# B&R Automation Studio project Teknologia25 (part 7)

### global.typ
```iecst
(*
Program: Robot

Description
(short summary)

*)
(*========== STATES ==========*)

TYPE
	RobotStateEnum :
		(
		ROBOT_INITIALIZE,
		ROBOT_IDLE,
		ROBOT_CMD_NORMAL,
		ROBOT_CMD_TARGET,
		ROBOT_COMMAND_DONE,
		ROBOT_COMMAND_ERROR,
		ROBOT_ERROR
		);
END_TYPE

(*========== INPUTS ==========*)

TYPE
	RobotInputCommandType : 	STRUCT
		Home : BOOL;
		PickUp : BOOL;
		GetCandy : BOOL;
		GiveCandy : BOOL;
		Dance : BOOL;
		HardReset : BOOL;
	END_STRUCT;
	RobotInputStatusType : 	STRUCT
		SetupComplete : BOOL;
	END_STRUCT;
	RobotInputType : 	STRUCT
		Force : BOOL;
		Command : RobotInputCommandType;
		Status : RobotInputStatusType;
		RobCommandNum : REAL;
		RobTargetX : REAL;
		RobTargetY : REAL;
	END_STRUCT;
END_TYPE

(*========== OUTPUTS ==========*)

TYPE
	RobotOutputCommandType : 	STRUCT
		NewCommand : BOOL;
	END_STRUCT;
	RobotOutputStatusType : 	STRUCT
		CommunicationOk : BOOL;
		CommandDone : BOOL;
		CommandError : BOOL;
		HardResetDone : BOOL;
		RobReady : BOOL;
		RobPhaseDone : BOOL;
		RobError : BOOL;
		RobPhaseNum : REAL;
		RobRapidState : BrAbbRwsStateRapidStateEnum;
		RobMotorState : BrAbbRwsStateMotorStateEnum;
		RobActiveMode : BrAbbRwsStateActiveModeEnum;
		ReadyForNextCommand : BOOL;
	END_STRUCT;
	RobotOutputType : 	STRUCT
		Command : RobotOutputCommandType;
		Status : RobotOutputStatusType;
	END_STRUCT;
END_TYPE

(*========== ERRORS ==========*)

TYPE
	RobotErrorType : 	STRUCT
		Active : BOOL;
		Acknowledge : BOOL;
		Code : DINT;
		Description : STRING[80];
	END_STRUCT;
END_TYPE

(*========== SETTINGS ==========*)

TYPE
	RobotSettingsType : 	STRUCT
		Enable : BOOL;
	END_STRUCT;
END_TYPE

(*========== INTERFACE ==========*)

TYPE
	RobotType : 	STRUCT
		Error : RobotErrorType;
		Input : RobotInputType;
		Output : RobotOutputType;
		Settings : RobotSettingsType;
		IsSimulated : BOOL;
		State : RobotStateEnum;
		SubState : DINT;
		StateInfo : STRING[255];
		OnStateEntry : BOOL; (*True for one cycle after state change*)
		robReadState : DINT;
	END_STRUCT;
END_TYPE
```

### Program Logical/Robot/Robot (IEC)

#### Robot.st
```iecst
PROGRAM _INIT

    // Access the task interface
	task ACCESS ADR(gRobot);

	// Check for simulator
	task.IsSimulated := DiagCpuIsSimulated();

	fb.BrAbbRwsCore_0.Parameters.UserName := 'Admin';
	fb.BrAbbRwsCore_0.Parameters.Password := 'robotics';
	fb.BrAbbRwsCore_0.Parameters.WebServerVersion := BR_ABB_RWS_VERSION_V2;
	fb.BrAbbRwsCore_0.Parameters.HostPort := 443;
	fb.BrAbbRwsCore_0.Parameters.Timeout := 0;
	fb.BrAbbRwsCore_0.Parameters.SecureConfigName := 'mySSLConfig';

	IF DiagCpuIsSimulated() THEN
		fb.BrAbbRwsCore_0.Parameters.ServerIP := '127.0.0.1';
	ELSE
		fb.BrAbbRwsCore_0.Parameters.ServerIP := '192.168.125.1';
	END_IF;

	fb.BrAbbRwsVariable_read.Parameters.Module := 'TeknologiaDemo25';
	fb.BrAbbRwsVariable_read.Parameters.Task := 'T_ROB1';
	fb.BrAbbRwsVariable_write.Parameters.Module := 'TeknologiaDemo25';
	fb.BrAbbRwsVariable_write.Parameters.Task := 'T_ROB1';

END_PROGRAM

PROGRAM _CYCLIC

    // Access task interface
    // =================================================================================================================
    task ACCESS ADR(gRobot);

    // Inputs
    // =================================================================================================================
    IF NOT task.Input.Force THEN
		task.Input.Command.Home := gMain.Output.Command.robHome;
		task.Input.Command.GetCandy := gMain.Output.Command.robGetPrize;
		task.Input.Command.Dance := gMain.Output.Command.robDance;
		task.Input.Command.GiveCandy := gMain.Output.Command.robGivePrize;
		task.Input.Command.PickUp := gMain.Output.Command.robPickup;
	END_IF

	task.Error.Active := fb.BrAbbRwsCore_0.Error OR fb.BrAbbRwsGetState_0.Error;

    // Task state machine
    // =================================================================================================================
    CASE task.State OF
        ROBOT_INITIALIZE:
			CASE task.SubState OF
				0:
					task.StateInfo := 'Initializing';
					// ---------------------------------------------------------------------------------
					fb.BrAbbRwsCore_0.Enable := FALSE;
					brsmemset(ADR(local), 0, SIZEOF(local));
					task.SubState := 10;
				10:
					task.StateInfo := 'Connecting to robot';
					// ---------------------------------------------------------------------------------
					fb.BrAbbRwsCore_0.Enable := TRUE;

					IF fb.BrAbbRwsCore_0.Active THEN
						task.State := ROBOT_IDLE;
						fb.BrAbbRwsGetState_0.Ident := fb.BrAbbRwsCore_0.Ident;
						fb.BrAbbRwsVariable_read.Ident := fb.BrAbbRwsCore_0.Ident;
						fb.BrAbbRwsVariable_write.Ident := fb.BrAbbRwsCore_0.Ident;
						local.readRobotValues := TRUE;
						fb.BrAbbRwsVariable_write.Enable := TRUE;
					ELSIF fb.BrAbbRwsCore_0.Error THEN
						task.Error.Code := fb.BrAbbRwsCore_0.StatusID;
						task.SubState := 30;
					END_IF;
			END_CASE;

		ROBOT_IDLE:
			task.StateInfo := 'Ready for commands';
			// ---------------------------------------------------------------------------------
			IF task.Input.Command.Home THEN
				task.Input.RobCommandNum := 1;
				task.State := ROBOT_CMD_NORMAL;

			ELSIF task.Input.Command.Dance THEN
				task.Input.RobCommandNum := 3;
				task.State := ROBOT_CMD_NORMAL;

			ELSIF task.Input.Command.GetCandy THEN
				task.Input.RobCommandNum := 4;
				task.State := ROBOT_CMD_NORMAL;

			ELSIF task.Input.Command.PickUp THEN
				task.Input.RobCommandNum := 2;
				task.State := ROBOT_CMD_TARGET;

			ELSIF task.Input.Command.GiveCandy THEN
				task.Input.RobCommandNum := 5;
				task.State := ROBOT_CMD_TARGET;
			END_IF;

		ROBOT_CMD_NORMAL:
			CASE task.SubState OF
				0:
					task.StateInfo := 'Execute command';
					// ---------------------------------------------------------------------------------
					fb.BrAbbRwsVariable_write.Parameters.Variable := 'nAcoposCmd';
					fb.BrAbbRwsVariable_write.Value.DataAdress := ADR(task.Input.RobCommandNum);
					fb.BrAbbRwsVariable_write.Value.DataType := BR_ABB_RWS_VAR_NUM;

					local.actions.substate.write := TRUE;

					IF fb.BrAbbRwsVariable_write.Done THEN
	  					task.SubState := 10;
					ELSIF fb.BrAbbRwsVariable_write.Error THEN
						task.State := ROBOT_COMMAND_ERROR;
					END_IF;

				10:
					task.StateInfo := 'Wait robot to complete';
					// ---------------------------------------------------------------------------------
					IF task.Output.Status.RobPhaseDone THEN
						task.SubState := 20;
					END_IF;

				20:
					task.StateInfo := 'Reset robot command';
					// ---------------------------------------------------------------------------------
					task.Input.RobCommandNum := 0;

					fb.BrAbbRwsVariable_write.Parameters.Variable := 'nAcoposCmd';
					fb.BrAbbRwsVariable_write.Value.DataAdress := ADR(task.Input.RobCommandNum);
					fb.BrAbbRwsVariable_write.Value.DataType := BR_ABB_RWS_VAR_NUM;

					local.actions.substate.write := TRUE;

					IF fb.BrAbbRwsVariable_write.Done THEN
						task.State := ROBOT_COMMAND_DONE;
					ELSIF fb.BrAbbRwsVariable_write.Error THEN
						task.State := ROBOT_COMMAND_ERROR;
					END_IF;
			END_CASE;

		ROBOT_CMD_TARGET:
			CASE task.SubState OF
				0:
					task.StateInfo := 'Write X';
					// ---------------------------------------------------------------------------------
					local.robTargetX_mm := 1000 * task.Input.RobTargetX;

					fb.BrAbbRwsVariable_write.Parameters.Variable := 'nPos_X';
					fb.BrAbbRwsVariable_write.Value.DataAdress := ADR(local.robTargetX_mm);
					fb.BrAbbRwsVariable_write.Value.DataType := BR_ABB_RWS_VAR_NUM;

					local.actions.substate.write := TRUE;

					IF fb.BrAbbRwsVariable_write.Done THEN
						task.SubState := 10;
					ELSIF fb.BrAbbRwsVariable_write.Error THEN
						task.State := ROBOT_COMMAND_ERROR;
					END_IF;

				10:
					task.StateInfo := 'Write Y';
					// ---------------------------------------------------------------------------------
					local.robTargetY_mm := 1000 * task.Input.RobTargetY;

					fb.BrAbbRwsVariable_write.Parameters.Variable := 'nPos_Y';
					fb.BrAbbRwsVariable_write.Value.DataAdress := ADR(local.robTargetY_mm);
					fb.BrAbbRwsVariable_write.Value.DataType := BR_ABB_RWS_VAR_NUM;

					local.actions.substate.write := TRUE;

					IF fb.BrAbbRwsVariable_write.Done THEN
						task.SubState := 20;
					ELSIF fb.BrAbbRwsVariable_write.Error THEN
						task.State := ROBOT_COMMAND_ERROR;
					END_IF;

				20:
					task.StateInfo := 'Write command num';
					// ---------------------------------------------------------------------------------
					fb.BrAbbRwsVariable_write.Parameters.Variable := 'nAcoposCmd';
					fb.BrAbbRwsVariable_write.Value.DataAdress := ADR(task.Input.RobCommandNum);
					fb.BrAbbRwsVariable_write.Value.DataType := BR_ABB_RWS_VAR_NUM;

					local.actions.substate.write := TRUE;

					IF fb.BrAbbRwsVariable_write.Done THEN
						task.SubState := 30;
					ELSIF fb.BrAbbRwsVariable_write.Error THEN
						task.State := ROBOT_COMMAND_ERROR;
					END_IF;

				30:
					task.StateInfo := 'Wait robot to complete';
					// ---------------------------------------------------------------------------------
					IF task.Output.Status.RobPhaseDone THEN
						task.SubState := 40;
					END_IF;

				40:
					task.StateInfo := 'Reset robot command';
					// ---------------------------------------------------------------------------------
					task.Input.RobCommandNum := 0;

					fb.BrAbbRwsVariable_write.Parameters.Variable := 'nAcoposCmd';
					fb.BrAbbRwsVariable_write.Value.DataAdress := ADR(task.Input.RobCommandNum);
					fb.BrAbbRwsVariable_write.Value.DataType := BR_ABB_RWS_VAR_NUM;

					local.actions.substate.write := TRUE;

					IF fb.BrAbbRwsVariable_write.Done THEN
						task.State := ROBOT_COMMAND_DONE;
					ELSIF fb.BrAbbRwsVariable_write.Error THEN
						task.State := ROBOT_COMMAND_ERROR;
					END_IF;
			END_CASE;

		ROBOT_COMMAND_DONE:
			task.StateInfo := 'Command done';
			// ---------------------------------------------------------------------------------
			local.actions.substate.command_done := TRUE;

			IF brsmemcmp(ADR(task.Input.Command), ADR(no_command), SIZEOF(no_command)) = 0 THEN
				task.State := ROBOT_IDLE;
			END_IF;

		ROBOT_COMMAND_ERROR:
			task.StateInfo := 'Command error';
			// ---------------------------------------------------------------------------------
			local.actions.substate.command_error := TRUE;
			local.actions.substate.write_reset := TRUE;

			IF brsmemcmp(ADR(task.Input.Command), ADR(no_command), SIZEOF(no_command)) = 0 THEN
				task.State := ROBOT_IDLE;
			END_IF;

		ROBOT_ERROR:
			// Error occured during execution
            // ---------------------------------------------------------------------------------
            IF task.Error.Acknowledge THEN
                brsmemset(ADR(task.Error), 0, SIZEOF(task.Error));
                task.State := ROBOT_INITIALIZE;
            END_IF;
    END_CASE // End of main task logic

    task.Error.Acknowledge := FALSE;

    // Detect state change events
    // =================================================================================================================
    task.OnStateEntry := (task.State <> local.lastState) OR (task.SubState <> local.lastSubState);

    IF task.State <> local.lastState THEN
        task.SubState := 0;
        local.lastState := task.State;
        brsmemset(ADR(local.actions.state), 0, SIZEOF(local.actions.state));
		brsmemset(ADR(local.actions.substate), 0, SIZEOF(local.actions.substate));
		task.StateInfo := '';
    END_IF

    // Reset current state actions also when substate changes
    IF task.SubState <> local.lastSubState THEN
        local.lastSubState := task.SubState;
		brsmemset(ADR(local.actions.substate), 0, SIZEOF(local.actions.substate));
		task.StateInfo := '';
    END_IF

	// Robot state poll
	// =================================================================================================================
	CASE task.robReadState OF
		0:
			// ---------------------------------------------------------------------------------
			IF local.readRobotValues THEN
				fb.BrAbbRwsGetState_0.Enable := TRUE;
				fb.BrAbbRwsVariable_read.Enable := TRUE;

				IF fb.BrAbbRwsGetState_0.Active AND fb.BrAbbRwsVariable_read.Active THEN

					task.robReadState := 10;
					local.robReadNum := 0;
				END_IF;
			END_IF;

		10:
			// ---------------------------------------------------------------------------------
			fb.TON_ReadDelay.IN := TRUE;
			fb.TON_ReadDelay.PT := T#20ms;

			IF local.readRobotValues = FALSE THEN
				task.robReadState := 0;
			ELSIF fb.TON_ReadDelay.Q THEN
				fb.TON_ReadDelay.IN := FALSE;
				task.robReadState := 100 + local.robReadNum;
				local.robReadNum := local.robReadNum + 1;
			END_IF;

		50:
			// ---------------------------------------------------------------------------------
			fb.TON_ReadDelay.IN := TRUE;
			fb.TON_ReadDelay.PT := T#2s;

			task.Output.Status.CommunicationOk := FALSE;

			fb.BrAbbRwsGetState_0.Enable := FALSE;
			fb.BrAbbRwsVariable_read.Enable := FALSE;

			IF fb.TON_ReadDelay.Q THEN
				fb.TON_ReadDelay.IN := FALSE;
				IF fb.BrAbbRwsCore_0.Error THEN
	  				task.robReadState := 60;
				ELSE
					task.robReadState := 0;
				END_IF;
			END_IF;

		60:
			// ---------------------------------------------------------------------------------
			fb.BrAbbRwsCore_0.ErrorReset := TRUE;

			IF NOT fb.BrAbbRwsCore_0.Error THEN
				fb.BrAbbRwsCore_0.ErrorReset := FALSE;
				task.robReadState := 0;
			END_IF;

		100:
			// ---------------------------------------------------------------------------------
			fb.BrAbbRwsGetState_0.Parameters.MechUnit := 'ROB1';
			fb.BrAbbRwsGetState_0.Parameters.Enable.ActPosCart := FALSE;
			fb.BrAbbRwsGetState_0.GetState := TRUE;

			IF fb.BrAbbRwsGetState_0.Done THEN
				task.Output.Status.CommunicationOk := TRUE;
				task.Output.Status.RobRapidState := fb.BrAbbRwsGetState_0.RapidState;
				task.Output.Status.RobMotorState := fb.BrAbbRwsGetState_0.MotorState;
				task.Output.Status.RobActiveMode := fb.BrAbbRwsGetState_0.ActiveMode;
				task.robReadState := 10;
			ELSIF fb.BrAbbRwsGetState_0.Error THEN
				task.Output.Status.RobRapidState := fb.BrAbbRwsGetState_0.RapidState;
				task.Output.Status.RobMotorState := fb.BrAbbRwsGetState_0.MotorState;
				task.Output.Status.RobActiveMode := fb.BrAbbRwsGetState_0.ActiveMode;
				task.robReadState := 50;
			END_IF;

		101:
			// ---------------------------------------------------------------------------------
			fb.BrAbbRwsVariable_read.Parameters.Variable := 'bRobotPhaseDone';
			fb.BrAbbRwsVariable_read.Value.DataAdress := ADR(gRobot.Output.Status.RobPhaseDone);
			fb.BrAbbRwsVariable_read.Value.DataType := BR_ABB_RWS_VAR_BOOL;
			fb.BrAbbRwsVariable_read.GetValue := TRUE;

			IF fb.BrAbbRwsVariable_read.Done THEN
				task.robReadState := 10;
			ELSIF fb.BrAbbRwsVariable_read.Error THEN
				task.robReadState := 50;
			END_IF;

		102:
			// ---------------------------------------------------------------------------------
			fb.BrAbbRwsVariable_read.Parameters.Variable := 'bRobotReady';
			fb.BrAbbRwsVariable_read.Value.DataAdress := ADR(gRobot.Output.Status.RobReady);
			fb.BrAbbRwsVariable_read.Value.DataType := BR_ABB_RWS_VAR_BOOL;
			fb.BrAbbRwsVariable_read.GetValue := TRUE;

			IF fb.BrAbbRwsVariable_read.Done THEN
				task.robReadState := 10;
			ELSIF fb.BrAbbRwsVariable_read.Error THEN
				task.robReadState := 50;
			END_IF;

		103:
			// ---------------------------------------------------------------------------------
			fb.BrAbbRwsVariable_read.Parameters.Variable := 'bRobotError';
			fb.BrAbbRwsVariable_read.Value.DataAdress := ADR(gRobot.Output.Status.RobError);
			fb.BrAbbRwsVariable_read.Value.DataType := BR_ABB_RWS_VAR_BOOL;
			fb.BrAbbRwsVariable_read.GetValue := TRUE;

			IF fb.BrAbbRwsVariable_read.Done THEN
				task.robReadState := 10;
			ELSIF fb.BrAbbRwsVariable_read.Error THEN
				task.robReadState := 50;
			END_IF;

		104:
			// ---------------------------------------------------------------------------------
			fb.BrAbbRwsVariable_read.Parameters.Variable := 'nRobotPhase';
			fb.BrAbbRwsVariable_read.Value.DataAdress := ADR(gRobot.Output.Status.RobPhaseNum);
			fb.BrAbbRwsVariable_read.Value.DataType := BR_ABB_RWS_VAR_NUM;
			fb.BrAbbRwsVariable_read.GetValue := TRUE;

			IF fb.BrAbbRwsVariable_read.Done THEN
				task.robReadState := 1000;
			ELSIF fb.BrAbbRwsVariable_read.Error THEN
				task.robReadState := 50;
			END_IF;

		1000:
			task.robReadState := 10;
			local.robReadNum := 0;
	END_CASE;

	IF task.robReadState <> local.robReadStateLast THEN
		local.robReadStateLast := task.robReadState;
		fb.BrAbbRwsGetState_0.GetState := FALSE;
		fb.BrAbbRwsVariable_read.GetValue := FALSE;
		fb.BrAbbRwsVariable_read.SetValue := FALSE;
		fb.BrAbbRwsVariable_read.SetValue := FALSE;
	END_IF;

    // Function calls
    // =================================================================================================================
    fb.BrAbbRwsCore_0();
	fb.TON_ReadDelay();
	fb.BrAbbRwsGetState_0();
	fb.BrAbbRwsVariable_read();

	fb.BrAbbRwsVariable_write.SetValue := local.actions.substate.write;
	fb.BrAbbRwsVariable_write.ErrorReset := local.actions.substate.write_reset;
	fb.BrAbbRwsVariable_write();

    // Task outputs
    // =================================================================================================================
	task.Output.Status.CommandDone := local.actions.substate.command_done;
	task.Output.Status.CommandError := local.actions.substate.command_error;

END_PROGRAM

PROGRAM _EXIT

//	WHILE fb.BrAbbRwsGetState_0.Active DO
//		fb.BrAbbRwsGetState_0(Enable := FALSE);
//	END_WHILE
//
//	WHILE fb.BrAbbRwsVariable_read.Active DO
//		fb.BrAbbRwsVariable_read(Enable := FALSE);
//	END_WHILE
//
//	task.robReadState := 100;
//	task.robReadState := 0;

END_PROGRAM
```

#### local.typ
```iecst
TYPE
	RobotFbType : 	STRUCT
		BrAbbRwsCore_0 : BrAbbRwsCore;
		BrAbbRwsVariable_read : BrAbbRwsVariable;
		BrAbbRwsVariable_write : BrAbbRwsVariable;
		BrAbbRwsGetState_0 : BrAbbRwsGetState;
		TON_RobState : TON;
		TON_ReadDelay : TON;
	END_STRUCT;
	RobotLocalType : 	STRUCT
		lastState : DINT;
		lastSubState : DINT;
		actions : RobotActionsType;
		readRobotValues : BOOL;
		robReadStateLast : DINT;
		robReadNum : DINT;
		robTargetX_mm : REAL;
		robTargetY_mm : REAL;
	END_STRUCT;
	RobotActionsType : 	STRUCT
		task : RobotTaskActionsType; (*Task actions are not automatically reset*)
		state : RobotStateActionsType; (*State actions are automatically reset whenever major task changes*)
		substate : RobotSubstateActionsType; (*Substate actions are automatically reset whenever major or substate changes*)
	END_STRUCT;
	RobotTaskActionsType : 	STRUCT
		task_action : BOOL;
	END_STRUCT;
	RobotStateActionsType : 	STRUCT
		state_action : BOOL;
	END_STRUCT;
	RobotSubstateActionsType : 	STRUCT
		command_done : BOOL;
		command_error : BOOL;
		write : BOOL;
		write_reset : BOOL;
	END_STRUCT;
	RobotHmiType : 	STRUCT
		isRunning : BOOL;
	END_STRUCT;
END_TYPE
```

#### local.var
```iecst
VAR
	task : REFERENCE TO RobotType;
	local : RobotLocalType;
	fb : RobotFbType;
	hmi : RobotHmiType;
	no_command : RobotInputCommandType;
END_VAR
```

- Visualisation Logical/mappView (not shown)

### Program Logical/Acp6D1 (IEC)

#### Acp6D.st
```iecst
PROGRAM _INIT

    // Access the task interface
	task ACCESS ADR(gAcp6D);

	// Check for simulator
	task.IsSimulated := DiagCpuIsSimulated();

	gCommInput;
	gCommOutput;
	gAssembly6D_1;

	// Fill in index of the shuttle element for easier access later on
	FOR i:=0 TO gMAX_INDEX_SHUTTLE DO
		local.shuttleOrder[i] := DINT_TO_UINT(i);
	END_FOR;

	acInitializePositions;

	moveQueueParamDefault.acceleration := 15.0;
	moveQueueParamDefault.acceleration_rotary := 0.1;
	moveQueueParamDefault.velocity_rotary := 0.1;
	moveQueueParamDefault.velocity_short := 0.1;
	moveQueueParamDefault.velocity_xy := 2.0;

	FOR i := 0 TO gMAX_INDEX_SHUTTLE DO
		fb.MoveQueue[i].Parameters := moveQueueParamDefault;
	END_FOR;

	// soundwave liikerata
	// Victory dance logiikka aalto z-aalto aalto -> vanhoihin asemmin -> keskellä spin ja z pomppuja -> kehällä arc movella kiertoradalle ja muutamak ierros ympäri -> paririviin keinahtelemaan ja kumartamaan pelaajalle
	// pelilogiikka mainiin
	// warm restartg mainiin
	// pelikäyttöliittymäsekvenssi
	// Circular shuffle loppuun -> group -> arc move -> sun planet -> asyncillä user selectiin
	// group fbt ja komennot
	// sun plenet tarkistus ja fb

END_PROGRAM

PROGRAM _CYCLIC
    // Access task interface
    // =================================================================================================================
	task ACCESS ADR(gAcp6D);

	test.SunShuttle := ADR(shuttles[4].Ref);
	test.PlanetShuttles[0] := shuttles[3].Ref;
	test();

	// Inputs
	// =================================================================================================================
	IF NOT task.Input.Force THEN
		task.Input.Command.MoveTo.Home := gMain.Output.Command.br6dHome;
		task.Input.Command.Shuffle.Circular := gMain.Output.Command.br6dcircularShuffle;
		task.Input.Command.FindPayload := gMain.Output.Command.br6dFindPayload;
		task.Input.Command.Victory := gMain.Output.Command.br6dLoseDance;
		task.Input.Command.ForceReset := gMain.Output.Command.br6dReset;
		task.Input.Command.SelectShuttle := gMain.Output.Command.br6dSelectShuttle;
		task.Input.Command.Shuffle.Simple := gMain.Output.Command.br6dSimpleShuffle;
		task.Input.Command.Victory := gMain.Output.Command.br6dWinDance;
	END_IF

	// Task state machine
	// =================================================================================================================
	CASE task.State OF
		ACP6D_INITIALIZE:
			CASE task.SubState OF
				0:
					task.StateInfo := 'Wait assembly to boot up';
					// ---------------------------------------------------------------------------------
					local.actions.state.cyclicModeRequest := a6dCYCLIC_DISABLED;

					fb.AssemblyReadInfo.Enable := TRUE;
					//Wait for the startup phase to be finished
					IF fb.AssemblyReadInfo.Valid THEN
						IF (fb.AssemblyReadInfo.AssemblyInfo.AssemblyState = mcACP6D_ERRORSTOP) THEN
							task.State := ACP6D_ERROR;
						ELSIF (fb.AssemblyReadInfo.AssemblyInfo.AssemblyState <> mcACP6D_STARTUP) THEN
							task.SubState := 10;
						END_IF
					END_IF

				10:
					task.StateInfo := 'Power off assembly';
					// ---------------------------------------------------------------------------------
					local.actions.substate.assemblyPowerOff := TRUE;

					IF fb.AssemblyPowerOff.Done THEN
						task.SubState := 20;
					ELSIF fb.AssemblyPowerOff.Error THEN
						task.Error.Code := fb.AssemblyPowerOff.ErrorID;
						task.State := ACP6D_ERROR;
					END_IF

				20:
					task.StateInfo := 'Power on assembly';
					// ---------------------------------------------------------------------------------
					IF task.OnStateEntry THEN
						brsmemset(ADR(shuttles), 0, SIZEOF(shuttles));
					END_IF;

					local.actions.substate.assemblyPowerOn := TRUE;

					IF fb.AssemblyPowerOn.Done THEN
						task.SubState := 100;
					ELSIF fb.AssemblyPowerOn.Error THEN
						task.Error.Code := fb.AssemblyPowerOn.ErrorID;
						task.State := ACP6D_ERROR;
					END_IF

				100:
					task.StateInfo := 'Read shuttle info - Read';
					// ---------------------------------------------------------------------------------
					local.actions.state.assemblyGetShuttles := TRUE;

					IF fb.AssemblyGetShuttle.Valid THEN
						task.Output.TotalShuttleCount := fb.AssemblyGetShuttle.TotalCount;
						local.actions.state.assemblyGetNextShuttle := FALSE;

						IF (fb.AssemblyGetShuttle.TotalCount = 0) THEN
							task.SubState := 1000;
							RETURN;
						END_IF;

						// Read shuttle information
						// Prevent access to wrong memory area
						i := LIMIT(0, UINT_TO_DINT(fb.AssemblyGetShuttle.TotalCount - fb.AssemblyGetShuttle.RemainingCount - 1), gMAX_INDEX_SHUTTLE);

						shuttles[i].ID := fb.AssemblyGetShuttle.AdditionalInfo.ShuttleID;
						shuttles[i].Ref := fb.AssemblyGetShuttle.Shuttle;
						shuttles[i].index := i;

						task.SubState := 110;
					END_IF

				110:
					task.StateInfo := 'Read shuttle info - Get next';
					// ---------------------------------------------------------------------------------
					IF (fb.AssemblyGetShuttle.RemainingCount > 0) THEN
						local.actions.state.assemblyGetNextShuttle := TRUE;
						task.SubState := 100;
					ELSE
						IF local.virtualShuttleCount >= MAX_NUM_SHUTTLE_VIRTUAL THEN
	  						task.State := ACP6D_COMMAND_DONE;
						ELSE
							task.SubState := 200;
						END_IF;
					END_IF

				200:
					task.StateInfo := 'Create virtual shuttle';
					// ---------------------------------------------------------------------------------
					local.actions.substate.createShuttleVirtual := TRUE;

					IF fb.virtualShCreate.Done THEN
						shuttlesVirtual[local.virtualShuttleCount] := fb.virtualShCreate.VirtualShuttle;
						local.virtualShuttleCount := local.virtualShuttleCount + 1;
						task.SubState := 210;
					ELSIF fb.virtualShCreate.Error THEN
						task.Error.Code := fb.virtualShCreate.ErrorID;
						task.State := ACP6D_ERROR;
					END_IF

				210:
					task.StateInfo := 'Check if enough virtual shuttles have been created';
					// ---------------------------------------------------------------------------------
					IF local.virtualShuttleCount >= MAX_NUM_SHUTTLE_VIRTUAL THEN
						task.State := ACP6D_COMMAND_DONE;
					ELSE
						task.SubState := 200;
					END_IF;

				1000:
					task.StateInfo := 'No shuttles';
				// ---------------------------------------------------------------------------------

			END_CASE;

		ACP6D_IDLE:
			task.StateInfo := 'Waiting for command';
			task.Output.Status.Initialized := TRUE;

			IF task.Input.Command.Reinitialize THEN
				task.State := ACP6D_INITIALIZE;

			ELSIF task.Input.Command.StartDemoMode THEN
				task.State := ACP6D_DEMO;

			ELSIF task.Input.Command.FindPayload THEN
				task.State := ACP6D_FIND_PAYLOAD;

			ELSIF task.Input.Command.SelectShuttle THEN
				task.State := ACP6D_SELECT_SHUTTLE;

			ELSIF task.Input.Command.StopAll THEN
				task.State := ACP6D_STOP_ALL;

			ELSIF task.Input.Command.ForceReset THEN
				task.State := ACP6D_FORCE_RESET;

			ELSIF task.Input.Command.Victory THEN
				task.State := ACP6D_VICTORY;

			ELSIF task.Input.Command.Animate THEN
				task.State := ACP6D_ANIMATE;

				// Move commands
			ELSIF task.Input.Command.MoveTo.Home THEN
				local.targetPos := positions.home;
				task.State := ACP6D_MOVE_TO;

			ELSIF task.Input.Command.MoveTo.User THEN
				local.targetPos := positions.user;
				task.State := ACP6D_MOVE_TO;

			ELSIF task.Input.Command.MoveTo.Dance THEN
				local.targetPos := positions.dance;
				task.State := ACP6D_MOVE_TO;

			ELSIF task.Input.Command.MoveTo.Clockface THEN
				local.targetPos := positions.clockface;
				task.State := ACP6D_MOVE_TO;

			ELSIF task.Input.Command.MoveTo.Pickup THEN
				local.targetPos := positions.pickup;
				task.State := ACP6D_MOVE_TO;

			ELSIF task.Input.Command.MoveTo.Shuffle THEN
				local.targetPos := positions.shuffle;
				task.State := ACP6D_MOVE_TO;

			ELSIF task.Input.Command.MoveTo.Side THEN
				local.targetPos := positions.side;
				task.State := ACP6D_MOVE_TO;

			// Shuffle commands
			ELSIF task.Input.Command.Shuffle.Simple THEN
				task.State := ACP6D_SHUFFLE_SIMPLE;

			ELSIF task.Input.Command.Shuffle.Circular THEN
				task.State := ACP6D_SHUFFLE_CIRCULAR;
			END_IF;

		ACP6D_DEMO:
			task.StateInfo := 'Running Acopos 6D feature demo';
			// ---------------------------------------------------------------------------------
			IF task.Input.Command.StopDemoMode THEN
				/// ..... Tähän kohtaan sit oma käsittely ja kun on demo taas inaktiviisiena niin hyppy COMMAND_DONE stateen
//				//IF FEATUREMODE INACTIEV THEN
//					task.State := ACP6D_COMMAND_DONE;
//				END_IF
			END_IF;

			//task.Output.Status.DemoModeActive := // MIKÄLIE LOGIIKKA ET MILLON ON PÄÄLLÄ!

		ACP6D_STOP_ALL:
			task.StateInfo := 'Stopping all shuttles';
			// ---------------------------------------------------------------------------------
			local.actions.substate.assemblyStop := TRUE;

			IF fb.assemblyStop.Done THEN
				task.State := ACP6D_COMMAND_DONE;
			ELSIF fb.assemblyStop.Done THEN
				task.Error.Code := fb.assemblyStop.ErrorID;
				task.State := ACP6D_COMMAND_ERROR;
			END_IF;

		ACP6D_FORCE_RESET:
			task.StateInfo := 'Stopping all shuttles';
			// ---------------------------------------------------------------------------------
			local.actions.substate.assemblyStop := TRUE;

			IF fb.assemblyStop.Done THEN
				task.State := ACP6D_INITIALIZE;
			ELSIF fb.assemblyStop.Done THEN
				task.Error.Code := fb.assemblyStop.ErrorID;
				task.State := ACP6D_COMMAND_ERROR;
			END_IF;

		ACP6D_MOVE_TO:
			CASE task.SubState OF
				0:
					task.StateInfo := 'Make sure assembly in correct state';
					// ---------------------------------------------------------------------------------
					task.SubState := 10;

				10:
					task.StateInfo := 'Move shuttles to target position';
					// ---------------------------------------------------------------------------------
					IF task.OnStateEntry THEN
						brfiShuffle(ADR(local.shuttleOrder));

						// Configure shuttle targets
						fb.MoveInPlaneAsync.Parameters.Velocity := 2;
						fb.MoveInPlaneAsync.Parameters.Acceleration := 15;

						fb.MoveInPlaneAsync.Parameters.Mode := mcACP6D_SHUTTLE_SORTED;

						FOR i := 0 TO gMAX_INDEX_SHUTTLE DO
							x := local.shuttleOrder[i];

							fb.MoveInPlaneAsync.Parameters.AsyncPar[i].Shuttle := ADR(shuttles[i].Ref);
							fb.MoveInPlaneAsync.Parameters.AsyncPar[x].X := local.targetPos[i].X;
							fb.MoveInPlaneAsync.Parameters.AsyncPar[x].Y := local.targetPos[i].Y;
						END_FOR;
					END_IF;

					local.actions.substate.moveInPlaneAsync := TRUE;

					IF fb.MoveInPlaneAsync.Done THEN
						task.State := ACP6D_COMMAND_DONE;
					ELSIF fb.MoveInPlaneAsync.Error THEN
						task.Error.Code := fb.MoveInPlaneAsync.ErrorID;
						task.State := ACP6D_COMMAND_ERROR;
					END_IF;
			END_CASE;

		ACP6D_FIND_PAYLOAD:
			CASE task.SubState OF
				0:
					task.StateInfo := 'Initialize';
					// ---------------------------------------------------------------------------------
					// Wait a moment before starting the force reading process so the movement has totally stopped
					local.actions.substate.delay := TRUE;
					fb.TON_delay.PT := T#1s;

					local.actions.state.cyclicModeRequest := a6dCYCLIC_READ_FORCE;

					// Also wait until all force readings are valid
					IF fb.TON_delay.Q AND cyclic.allForceValuesValid THEN
						task.SubState := 20;
					END_IF;

				20:
					task.StateInfo := 'Calculcate average Fz for shuttles';
					// ---------------------------------------------------------------------------------
					IF task.OnStateEntry THEN
						local.measurement_index := 0;
						FOR i := 0 TO gMAX_INDEX_SHUTTLE DO
							shuttle ACCESS ADR(shuttles[i]);
							brsmemset(ADR(shuttle.force.readings), 0, SIZEOF(shuttle.force.readings));
						END_FOR;
					END_IF;

					// Check if enough measurements have been recorder already
					IF local.measurement_index >= gMAX_INDEX_MEASUREMENT THEN
						FOR i := 0 TO gMAX_INDEX_SHUTTLE DO
							shuttle ACCESS ADR(shuttles[i]);

							shuttle.force.Z_avg := 0;

							FOR x := 0 TO gMAX_INDEX_MEASUREMENT DO
								shuttle.force.Z_avg := shuttle.force.Z_avg + shuttle.force.readings[x].Fz;
							END_FOR;

							shuttle.force.Z_avg := shuttle.force.Z_avg / MEASUREMENT_COUNT;
						END_FOR;
						task.SubState := 30;

					ELSIF shuttles[0].force.readings[local.measurement_index].Fz <> fb.ReadCyclicForce[0].CyclicForce.Fz THEN
						// Wait for next new value until measurement index is increased
						// Assume all channels received updates when first index of the cyclic force function block has new values
						FOR i := 0 TO gMAX_INDEX_SHUTTLE DO
							// Record received force values
							shuttle ACCESS ADR(shuttles[i]);
							shuttle.force.readings[local.measurement_index] := fb.ReadCyclicForce[shuttle.index].CyclicForce;
						END_FOR;

						local.measurement_index := local.measurement_index + 1;
					END_IF;

				30:
					task.StateInfo := 'Find which shuttle holds the payload';
					// ---------------------------------------------------------------------------------
					IF task.OnStateEntry THEN
						local.Fz_highest := 0;
					END_IF;

					FOR i := 0 TO gMAX_INDEX_SHUTTLE DO
						shuttle ACCESS ADR(shuttles[i]);

						IF shuttle.force.Z_avg > local.Fz_highest THEN
							local.Fz_highest := shuttle.force.Z_avg;
							task.Output.ShuttleWithPayload.index := i;
						END_IF;
					END_FOR;

					task.SubState := 40;

				40:
					task.StateInfo := 'Indicate which has payload';
					// ---------------------------------------------------------------------------------
					shuttle ACCESS ADR(shuttles[task.Output.ShuttleWithPayload.index]);
					refMoveQueue ACCESS ADR(fb.MoveQueue[shuttle.index]);

					IF task.OnStateEntry THEN
						refMoveQueue.Parameters.acceleration := 10;
						refMoveQueue.Parameters.velocity_short := 0.02;
						refMoveQueue.Parameters.velocity_xy := 1.0;

						AddCommand6D_xyz(ADR(commandQueue), sZ, 0, 0, 0.001, 0, 0, 0, mcACP6D_MOVE_ABSOLUTE);
						AddCommand6D_xyz(ADR(commandQueue), sZ, 0, 0, 0.004, 0, 0, 0, mcACP6D_MOVE_ABSOLUTE);
						AddCommand6D_xyz(ADR(commandQueue), sZ, 0, 0, 0.001, 0, 0, 0, mcACP6D_MOVE_ABSOLUTE);
						AddCommand6D_xyz(ADR(commandQueue), sZ, 0, 0, 0.004, 0, 0, 0, mcACP6D_MOVE_ABSOLUTE);
						AddCommand6D_xyz(ADR(commandQueue), sZ, 0, 0, 0.001, 0, 0, 0, mcACP6D_MOVE_ABSOLUTE);
						AddCommand6D_xyz(ADR(commandQueue), sZ, 0, 0, 0.004, 0, 0, 0, mcACP6D_MOVE_ABSOLUTE);
						AddCommand6D_xyz(ADR(commandQueue), sZ, 0, 0, 0.001, 0, 0, 0, mcACP6D_MOVE_ABSOLUTE);
						AddCommand6D_xyz(ADR(commandQueue), sZ, 0, 0, 0.004, 0, 0, 0, mcACP6D_MOVE_ABSOLUTE);
						AddCommand6D_xyz(ADR(commandQueue), sZ, 0, 0, 0.001, 0, 0, 0, mcACP6D_MOVE_ABSOLUTE);
						AddCommand6D_xyz(ADR(commandQueue), sZ, 0, 0, 0.004, 0, 0, 0, mcACP6D_MOVE_ABSOLUTE);
						AddCommand6D_xyz(ADR(commandQueue), sZ, 0, 0, 0.001, 0, 0, 0, mcACP6D_MOVE_ABSOLUTE);

						refMoveQueue.Commands := commandQueue;
					END_IF;

					shuttle.command.moveQueue := TRUE;

					IF refMoveQueue.Done THEN
						task.State := ACP6D_COMMAND_DONE;
					ELSIF refMoveQueue.Error THEN
						task.Error.Code := refMoveQueue.ErrorID;
						task.State := ACP6D_COMMAND_ERROR;
					END_IF;
			END_CASE

		ACP6D_SELECT_SHUTTLE:
			CASE task.SubState OF
				0:
					task.StateInfo := 'Move shuttles to the front of the table';
					// ---------------------------------------------------------------------------------
					IF task.OnStateEntry THEN
						local.selectedCount := brfiShuttleSelect(ADR(shuttles), ADR(selected1), 0, 0.24, 1, 1);

						FOR i := 0 TO gMAX_INDEX_SHUTTLE DO
							fb.MoveQueue[i].Parameters.velocity_short := 0.05;
						END_FOR;

						AddCommand6D_wait(ADR(commandQueue), 0);

						AddCommand6D_xyz(ADR(commandQueue), sZ, 0, 0, 0.001, 0, 0, 0, mcACP6D_MOVE_ABSOLUTE);
						AddCommand6D_xyz(ADR(commandQueue), sZ, 0, 0, 0.004, 0, 0, 0, mcACP6D_MOVE_ABSOLUTE);
						AddCommand6D_xyz(ADR(commandQueue), sZ, 0, 0, 0.001, 0, 0, 0, mcACP6D_MOVE_ABSOLUTE);
						AddCommand6D_xyz(ADR(commandQueue), sZ, 0, 0, 0.004, 0, 0, 0, mcACP6D_MOVE_ABSOLUTE);
						AddCommand6D_xyz(ADR(commandQueue), sZ, 0, 0, 0.001, 0, 0, 0, mcACP6D_MOVE_ABSOLUTE);
						AddCommand6D_xyz(ADR(commandQueue), sZ, 0, 0, 0.004, 0, 0, 0, mcACP6D_MOVE_ABSOLUTE);
						AddCommand6D_xyz(ADR(commandQueue), sZ, 0, 0, 0.001, 0, 0, 0, mcACP6D_MOVE_ABSOLUTE);

						AddCommand6D_xy(ADR(commandQueue), sY, 0, 0.900, 0, 0, 0, pathDIRECT, 0, mcACP6D_MOVE_ABSOLUTE);

						AddCommand6D_xyz(ADR(commandQueue), sZ, 0, 0, 0.003, 0, 0.1, 0, mcACP6D_MOVE_ABSOLUTE);
						AddCommand6D_Rxyz(ADR(commandQueue), sRx, -0.03, 0, 0, 0.3, mcACP6D_MOVE_ABSOLUTE);
						AddCommand6D_Rxyz(ADR(commandQueue), sRx, 0.00, 0, 0, 0.3, mcACP6D_MOVE_ABSOLUTE);

						AddCommand6D_xyz(ADR(commandQueue), sZ, 0, 0, 0.001, 0, 0, 0, mcACP6D_MOVE_ABSOLUTE);

						IF local.selectedCount > 0 THEN
							FOR i := 0 TO local.selectedCount - 1 DO
								fb.MoveQueue[selected1[i].index].Commands := commandQueue;
								fb.MoveQueue[selected1[i].index].Commands[0].waitTime := random.delays[i];
								shuttles[selected1[i].index].command.moveQueue := TRUE;
							END_FOR;
						END_IF;
					END_IF;

					IF queueStatus.allDone THEN
						task.SubState := 10;
					ELSIF queueStatus.error THEN
						task.Error.Code := queueStatus.errorID;
						task.State := ACP6D_COMMAND_ERROR;
					END_IF;

				10:
					task.StateInfo := 'Say hello to the player';
					// ---------------------------------------------------------------------------------
					IF task.OnStateEntry THEN
	  					local.selectedCount := brfiShuttleSelect(ADR(shuttles), ADR(selected1), 1, 1, 0, 0.240 * 3);

						AddCommand6D_wait(ADR(commandQueue), 0);
						AddCommand6D_xyz(ADR(commandQueue), sZ, 0, 0, 0.001, 0, 0, 0, mcACP6D_MOVE_ABSOLUTE);
						AddCommand6D_xyz(ADR(commandQueue), sZ, 0, 0, 0.004, 0, 0, 0, mcACP6D_MOVE_ABSOLUTE);
						AddCommand6D_wait(ADR(commandQueue), 0.1);
						AddCommand6D_xyz(ADR(commandQueue), sZ, 0, 0, 0.001, 0, 0, 0, mcACP6D_MOVE_ABSOLUTE);

						IF local.selectedCount > 0 THEN
							FOR i := 0 TO local.selectedCount - 1 DO
								fb.MoveQueue[selected1[i].index].Parameters.velocity_short := 0.03;

								fb.MoveQueue[selected1[i].index].Commands := commandQueue;
								fb.MoveQueue[selected1[i].index].Commands[0].waitTime := i * 0.1;
								shuttles[selected1[i].index].command.moveQueue := TRUE;
							END_FOR;
						END_IF;
					END_IF;

					IF queueStatus.allDone THEN
						task.SubState := 20;
					ELSIF queueStatus.error THEN
						task.Error.Code := queueStatus.errorID;
						task.State := ACP6D_COMMAND_ERROR;
					END_IF;

				20:
					task.StateInfo := 'Start force reading';
					// ---------------------------------------------------------------------------------
					local.actions.state.cyclicModeRequest := a6dCYCLIC_READ_FORCE;

					IF cyclic.allForceValuesValid THEN
						task.SubState := 30;
					END_IF;

				30:
					task.StateInfo := 'Wait user to select shuttle';
					// ---------------------------------------------------------------------------------
					IF task.OnStateEntry THEN
						FOR i := 0 TO gMAX_INDEX_SHUTTLE DO
							shuttle ACCESS ADR(shuttles[i]);
							shuttle.force.Fz_baseline := shuttle.force.value.Fz;
						END_FOR;
					END_IF

					FOR i := 0 TO gMAX_INDEX_SHUTTLE DO
						shuttle ACCESS ADR(shuttles[i]);
						// Detect shuttle press from force increase over treshold from baseline
						IF shuttle.force.value.Fz > (shuttle.force.Fz_baseline + 3.0) THEN
							task.SubState := 40;
							task.Output.ShuttleUserSelected.index := i;
						END_IF;
					END_FOR;

				40:
					task.StateInfo := 'Move selected shuttle';
					// ---------------------------------------------------------------------------------
					IF task.OnStateEntry THEN
						shuttle ACCESS ADR(shuttles[task.Output.ShuttleUserSelected.index]);
						refMoveQueue ACCESS ADR(fb.MoveQueue[shuttle.index]);

						refMoveQueue.Parameters.velocity_xy := 1.5;
						refMoveQueue.Parameters.acceleration := 5.0;

						AddCommand6D_xy(ADR(commandQueue), sX + sY, 0.0, -0.2, 0.5, 0.5, 0, pathDIRECT, 0, mcACP6D_MOVE_RELATIVE);
						AddCommand6D_xy(ADR(commandQueue), sX + sY, positions.pickup[0].X, positions.pickup[0].Y, 0, 15, 0, pathDIRECT, 0, mcACP6D_MOVE_ABSOLUTE);

						refMoveQueue.Commands := commandQueue;

						shuttle.command.moveQueue := TRUE;
					END_IF;

					IF refMoveQueue.Done THEN
						task.SubState := 50;
					ELSIF refMoveQueue.Error THEN
						task.Error.Code := refMoveQueue.ErrorID;
						task.SubState := ACP6D_COMMAND_ERROR;
					END_IF;

				50:
					task.StateInfo := 'Move all other shuttles to pickup';
					// ---------------------------------------------------------------------------------
					IF task.OnStateEntry THEN
						// Configure shuttle targets
						fb.MoveInPlaneAsync.Parameters.Velocity := 2;
						fb.MoveInPlaneAsync.Parameters.Acceleration := 15;

						fb.MoveInPlaneAsync.Parameters.Mode := mcACP6D_SHUTTLE_UNSORTED;

						x := 1;

						FOR i := 0 TO gMAX_INDEX_SHUTTLE DO
							IF i <> task.Output.ShuttleUserSelected.index THEN
								fb.MoveInPlaneAsync.Parameters.AsyncPar[i].Shuttle := ADR(shuttles[i].Ref);
								fb.MoveInPlaneAsync.Parameters.AsyncPar[i].X := positions.pickup[x].X;
								fb.MoveInPlaneAsync.Parameters.AsyncPar[i].Y := positions.pickup[x].Y;
								x := x + 1;
							END_IF;
						END_FOR;
					END_IF;

					local.actions.substate.moveInPlaneAsync := TRUE;

					IF fb.MoveInPlaneAsync.Done THEN
						task.SubState := 100;
					ELSIF fb.MoveInPlaneAsync.Error THEN
						task.Error.Code := fb.MoveInPlaneAsync.ErrorID;
						task.State := ACP6D_COMMAND_ERROR;
					END_IF;

				100:
					task.StateInfo := 'Transfer back to reading position values';
					// ---------------------------------------------------------------------------------
					local.actions.state.cyclicModeRequest := a6dCYCLIC_READ_POSITION;

					IF cyclic.allPositionsValid THEN
						task.State := ACP6D_COMMAND_DONE;
					END_IF;

			END_CASE;

		ACP6D_SHUFFLE_SIMPLE:
			CASE task.SubState OF
				0:
					task.StateInfo := 'Move shuttles to start position';
					// ---------------------------------------------------------------------------------
					IF task.OnStateEntry THEN
						brfiShuffle(ADR(local.shuttleOrder));

						brsmemset(ADR(shuffle), 0, SIZEOF(shuffle));

						// Configure shuttle targets
						fb.MoveInPlaneAsync.Parameters.Velocity := 2;
						fb.MoveInPlaneAsync.Parameters.Acceleration := 15;

						fb.MoveInPlaneAsync.Parameters.Mode := mcACP6D_SHUTTLE_SORTED;

						FOR i := 0 TO gMAX_INDEX_SHUTTLE DO
							x := local.shuttleOrder[i];
							IF x = shuttles[task.Output.ShuttleWithPayload.index].index THEN
	  							shuffle.payloadPos := i;
							END_IF;

							fb.MoveInPlaneAsync.Parameters.AsyncPar[i].Shuttle := ADR(shuttles[x].Ref);
							fb.MoveInPlaneAsync.Parameters.AsyncPar[i].X := positions.shuffle_simple[i].X;
							fb.MoveInPlaneAsync.Parameters.AsyncPar[i].Y := positions.shuffle_simple[i].Y;
						END_FOR;

						shuffle.randNum := RandValueDINT(0, 3);

						IF shuffle.payloadPos > 3 THEN
							fb.MoveInPlaneAsync.Parameters.AsyncPar[shuffle.payloadPos].Shuttle := fb.MoveInPlaneAsync.Parameters.AsyncPar[shuffle.randNum].Shuttle;
							fb.MoveInPlaneAsync.Parameters.AsyncPar[shuffle.randNum].Shuttle := ADR(shuttles[task.Output.ShuttleWithPayload.index].Ref);
						END_IF;

					END_IF;

					local.actions.substate.moveInPlaneAsync := TRUE;

					IF fb.MoveInPlaneAsync.Done THEN
						task.SubState := 10;
					ELSIF fb.MoveInPlaneAsync.Error THEN
						task.Error.Code := fb.MoveInPlaneAsync.ErrorID;
						task.State := ACP6D_COMMAND_ERROR;
					END_IF;

				10:
					task.StateInfo := 'Prepare for shuffle';
					// ---------------------------------------------------------------------------------
					brfiShuttleSelect(ADR(shuttles), ADR(selected1), 0, 0.480, 1, 1);
					fb.MoveQueue[selected1[0].index].Parameters := moveQueueParamDefault;
					fb.MoveQueue[selected1[1].index].Parameters := moveQueueParamDefault;
					fb.MoveQueue[selected1[2].index].Parameters := moveQueueParamDefault;
					fb.MoveQueue[selected1[3].index].Parameters := moveQueueParamDefault;
					shuffle.sequence := random.shuffleSequence;
					task.SubState := 20;

				20:
					task.StateInfo := 'Select next shuffle sequence';
					// ---------------------------------------------------------------------------------
					IF shuffle.step > gMAX_INDEX_SHUFFLE THEN
						task.SubState := 200;
					ELSE
						shuffle.invertedMove := shuffle.sequence[shuffle.step] < 0;
						shuffle.invertedDirection := SEL(shuffle.invertedMove, 1, -1);
						task.SubState := 100 + ABS(shuffle.sequence[shuffle.step]);
						shuffle.step := shuffle.step + 1;
					END_IF;

				100:
					task.StateInfo := 'Sides shift rotate';
					// ---------------------------------------------------------------------------------
					IF task.OnStateEntry THEN
						brfiShuttleSelect(ADR(shuttles), ADR(selected1), 0, 0.480, 1, 1);

						IF shuffle.invertedMove THEN
							AddCommand6D_arcAngularCW(ADR(fb.MoveQueue[selected1[0].index].Commands),  0.12, 0, brmPI, 0, 10, 0, mcACP6D_MOVE_RELATIVE);
							AddCommand6D_arcAngularCW(ADR(fb.MoveQueue[selected1[1].index].Commands), -0.12, 0, brmPI, 0, 10, 0, mcACP6D_MOVE_RELATIVE);

							AddCommand6D_arcAngularCW(ADR(fb.MoveQueue[selected1[2].index].Commands), 0.12, 0, brmPI, 0, 10, 0, mcACP6D_MOVE_RELATIVE);
							AddCommand6D_arcAngularCW(ADR(fb.MoveQueue[selected1[3].index].Commands), -0.12, 0, brmPI, 0, 10, 0, mcACP6D_MOVE_RELATIVE);
						ELSE
							AddCommand6D_arcAngularCCW(ADR(fb.MoveQueue[selected1[0].index].Commands),  0.12, 0, brmPI, 0, 10, 0, mcACP6D_MOVE_RELATIVE);
							AddCommand6D_arcAngularCCW(ADR(fb.MoveQueue[selected1[1].index].Commands), -0.12, 0, brmPI, 0, 10, 0, mcACP6D_MOVE_RELATIVE);

							AddCommand6D_arcAngularCCW(ADR(fb.MoveQueue[selected1[2].index].Commands), 0.12, 0, brmPI, 0, 10, 0, mcACP6D_MOVE_RELATIVE);
							AddCommand6D_arcAngularCCW(ADR(fb.MoveQueue[selected1[3].index].Commands), -0.12, 0, brmPI, 0, 10, 0, mcACP6D_MOVE_RELATIVE);
						END_IF;
					END_IF;

					shuttles[selected1[0].index].command.moveQueue := TRUE;
					shuttles[selected1[1].index].command.moveQueue := TRUE;
					shuttles[selected1[2].index].command.moveQueue := TRUE;
					shuttles[selected1[3].index].command.moveQueue := TRUE;

					IF queueStatus.allDone THEN
						task.SubState := 20;
					ELSIF queueStatus.error THEN
						task.Error.Code := queueStatus.errorID;
						task.State := ACP6D_COMMAND_ERROR;
					END_IF;

				101:
					task.StateInfo := 'Mid shift rotate';
					// ---------------------------------------------------------------------------------
					IF task.OnStateEntry THEN
						brfiShuttleSelect(ADR(shuttles), ADR(selected1), 0, 0.480, 1, 1);

						IF shuffle.invertedMove THEN
							AddCommand6D_arcAngularCW(ADR(commandQueue), 2 * 0.24, 3 * 0.24, brmPI, 0, 10, 0, mcACP6D_MOVE_ABSOLUTE);

							fb.MoveQueue[selected1[1].index].Commands := commandQueue;
							fb.MoveQueue[selected1[2].index].Commands := commandQueue;
						ELSE
							AddCommand6D_arcAngularCCW(ADR(commandQueue), 2 * 0.24, 3 * 0.24, brmPI, 0, 10, 0, mcACP6D_MOVE_ABSOLUTE);

							fb.MoveQueue[selected1[1].index].Commands := commandQueue;
							fb.MoveQueue[selected1[2].index].Commands := commandQueue;
						END_IF;
					END_IF;

					shuttles[selected1[1].index].command.moveQueue := TRUE;
					shuttles[selected1[2].index].command.moveQueue := TRUE;

					IF queueStatus.allDone THEN
						task.SubState := 20;
					ELSIF queueStatus.error THEN
						task.Error.Code := queueStatus.errorID;
						task.State := ACP6D_COMMAND_ERROR;
					END_IF;

				102:
					task.StateInfo := 'Sides shift';
					// ---------------------------------------------------------------------------------
					IF task.OnStateEntry THEN
						brfiShuttleSelect(ADR(shuttles), ADR(selected1), 0, 0.480, 1, 1);

						AddCommand6D_xy(ADR(fb.MoveQueue[selected1[0].index].Commands), sX + sY, 0, shuffle.invertedDirection  * -0.120, 0, 0, 0, pathY_X, 0, mcACP6D_MOVE_RELATIVE);
						AddCommand6D_xy(ADR(fb.MoveQueue[selected1[0].index].Commands), sX + sY, 3 * 0.240, 0, 0, 0, 0, pathY_X, 0, mcACP6D_MOVE_RELATIVE);
						AddCommand6D_xy(ADR(fb.MoveQueue[selected1[0].index].Commands), sX + sY, 0, shuffle.invertedDirection * 0.120, 0, 0, 0, pathY_X, 0, mcACP6D_MOVE_RELATIVE);

						AddCommand6D_xy(ADR(fb.MoveQueue[selected1[3].index].Commands), sX + sY, 0, shuffle.invertedDirection  * 0.120, 0, 0, 0, pathY_X, 0, mcACP6D_MOVE_RELATIVE);
						AddCommand6D_xy(ADR(fb.MoveQueue[selected1[3].index].Commands), sX + sY, -3 * 0.240, 0, 0, 0, 0, pathY_X, 0, mcACP6D_MOVE_RELATIVE);
						AddCommand6D_xy(ADR(fb.MoveQueue[selected1[3].index].Commands), sX + sY, 0, shuffle.invertedDirection  * -0.120, 0, 0, 0, pathY_X, 0, mcACP6D_MOVE_RELATIVE);
					END_IF;

					shuttles[selected1[0].index].command.moveQueue := TRUE;
					shuttles[selected1[3].index].command.moveQueue := TRUE;

					IF queueStatus.allDone THEN
						task.SubState := 20;
					ELSIF queueStatus.error THEN
						task.Error.Code := queueStatus.errorID;
						task.State := ACP6D_COMMAND_ERROR;
					END_IF;

				103:
					task.StateInfo := 'Middle to outside shift';
					// ---------------------------------------------------------------------------------
					IF task.OnStateEntry THEN
						brfiShuttleSelect(ADR(shuttles), ADR(selected1), 0, 0.480, 1, 1);

						AddCommand6D_xy(ADR(fb.MoveQueue[selected1[0].index].Commands), sX + sY, 0.240, 0, 0, 0, 0, pathY_X, 0.00, mcACP6D_MOVE_RELATIVE);
						AddCommand6D_xy(ADR(fb.MoveQueue[selected1[3].index].Commands), sX + sY, -0.240, 0, 0, 0, 0, pathY_X, 0.00, mcACP6D_MOVE_RELATIVE);

						AddCommand6D_xy(ADR(fb.MoveQueue[selected1[1].index].Commands), sX + sY, 0, shuffle.invertedDirection * 0.120, 0, 0, 0, pathY_X, 0.00, mcACP6D_MOVE_RELATIVE);
						AddCommand6D_xy(ADR(fb.MoveQueue[selected1[1].index].Commands), sX + sY, -0.240, 0, 0, 0, 0, pathY_X, 0.00, mcACP6D_MOVE_RELATIVE);
						AddCommand6D_xy(ADR(fb.MoveQueue[selected1[1].index].Commands), sX + sY, 0, shuffle.invertedDirection * -0.120, 0, 0, 0, pathY_X, 0.00, mcACP6D_MOVE_RELATIVE);

						AddCommand6D_xy(ADR(fb.MoveQueue[selected1[2].index].Commands), sX + sY, 0, shuffle.invertedDirection * 0.120, 0, 0, 0, pathY_X, 0.00, mcACP6D_MOVE_RELATIVE);
						AddCommand6D_xy(ADR(fb.MoveQueue[selected1[2].index].Commands), sX + sY, 0.240, 0, 0, 0, 0, pathY_X, 0.00, mcACP6D_MOVE_RELATIVE);
						AddCommand6D_xy(ADR(fb.MoveQueue[selected1[2].index].Commands), sX + sY, 0, shuffle.invertedDirection * -0.120, 0, 0, 0, pathY_X, 0.00, mcACP6D_MOVE_RELATIVE);
					END_IF;

					shuttles[selected1[0].index].command.moveQueue := TRUE;
					shuttles[selected1[1].index].command.moveQueue := TRUE;
					shuttles[selected1[2].index].command.moveQueue := TRUE;
					shuttles[selected1[3].index].command.moveQueue := TRUE;

					IF queueStatus.allDone THEN
						task.SubState := 20;
					ELSIF queueStatus.error THEN
						task.Error.Code := queueStatus.errorID;
						task.State := ACP6D_COMMAND_ERROR;
					END_IF;

				104:
					task.StateInfo := 'Twin shift';
					// ---------------------------------------------------------------------------------
					IF task.OnStateEntry THEN
						brfiShuttleSelect(ADR(shuttles), ADR(selected1), 0, 0.480, 1, 1);

						AddCommand6D_xy(ADR(fb.MoveQueue[selected1[0].index].Commands), sX + sY, 0, shuffle.invertedDirection * 0.120, 0, 0, 0, pathY_X, 0.00, mcACP6D_MOVE_RELATIVE);
						AddCommand6D_xy(ADR(fb.MoveQueue[selected1[2].index].Commands), sX + sY, 0, shuffle.invertedDirection * 0.120, 0, 0, 0, pathY_X, 0.00, mcACP6D_MOVE_RELATIVE);
						AddCommand6D_xy(ADR(fb.MoveQueue[selected1[0].index].Commands), sX + sY, 0.240, 0, 0, 0, 0, pathY_X, 0.00, mcACP6D_MOVE_RELATIVE);
						AddCommand6D_xy(ADR(fb.MoveQueue[selected1[2].index].Commands), sX + sY, 0.240, 0, 0, 0, 0, pathY_X, 0.00, mcACP6D_MOVE_RELATIVE);
						AddCommand6D_xy(ADR(fb.MoveQueue[selected1[0].index].Commands), sX + sY, 0, shuffle.invertedDirection * -0.120, 0, 0, 0, pathY_X, 0.00, mcACP6D_MOVE_RELATIVE);
						AddCommand6D_xy(ADR(fb.MoveQueue[selected1[2].index].Commands), sX + sY, 0, shuffle.invertedDirection * -0.120, 0, 0, 0, pathY_X, 0.00, mcACP6D_MOVE_RELATIVE);

						AddCommand6D_xy(ADR(fb.MoveQueue[selected1[1].index].Commands), sX + sY, 0, shuffle.invertedDirection * -0.120, 0, 0, 0, pathY_X, 0.00, mcACP6D_MOVE_RELATIVE);
						AddCommand6D_xy(ADR(fb.MoveQueue[selected1[3].index].Commands), sX + sY, 0, shuffle.invertedDirection * -0.120, 0, 0, 0, pathY_X, 0.00, mcACP6D_MOVE_RELATIVE);
						AddCommand6D_xy(ADR(fb.MoveQueue[selected1[1].index].Commands), sX + sY, -0.240, 0, 0, 0, 0, pathY_X, 0.00, mcACP6D_MOVE_RELATIVE);
						AddCommand6D_xy(ADR(fb.MoveQueue[selected1[3].index].Commands), sX + sY, -0.240, 0, 0, 0, 0, pathY_X, 0.00, mcACP6D_MOVE_RELATIVE);
						AddCommand6D_xy(ADR(fb.MoveQueue[selected1[1].index].Commands), sX + sY, 0, shuffle.invertedDirection * 0.120, 0, 0, 0, pathY_X, 0.00, mcACP6D_MOVE_RELATIVE);
						AddCommand6D_xy(ADR(fb.MoveQueue[selected1[3].index].Commands), sX + sY, 0, shuffle.invertedDirection * 0.120, 0, 0, 0, pathY_X, 0.00, mcACP6D_MOVE_RELATIVE);
					END_IF;

					shuttles[selected1[0].index].command.moveQueue := TRUE;
					shuttles[selected1[1].index].command.moveQueue := TRUE;
					shuttles[selected1[2].index].command.moveQueue := TRUE;
					shuttles[selected1[3].index].command.moveQueue := TRUE;

					IF queueStatus.allDone THEN
						task.SubState := 20;
					ELSIF queueStatus.error THEN
						task.Error.Code := queueStatus.errorID;
						task.State := ACP6D_COMMAND_ERROR;
					END_IF;

				200:
					task.StateInfo := 'Star shift 1';
					// ---------------------------------------------------------------------------------
					IF task.OnStateEntry THEN
						brfiShuttleSelect(ADR(shuttles), ADR(selected1), 0, 0.480, 1, 1);

						AddCommand6D_xy(ADR(fb.MoveQueue[selected1[0].index].Commands), sX + sY,  0.360, 0.140, 0, 0, 0, pathY_X, 0.00, mcACP6D_MOVE_RELATIVE);
						AddCommand6D_xy(ADR(fb.MoveQueue[selected1[3].index].Commands), sX + sY,  -0.360, -0.140, 0, 0, 0, pathY_X, 0.00, mcACP6D_MOVE_RELATIVE);

						AddCommand6D_xy(ADR(fb.MoveQueue[selected1[1].index].Commands), sX + sY,  -0.020, 0, 0, 0, 0, pathY_X, 0.00, mcACP6D_MOVE_RELATIVE);
						AddCommand6D_xy(ADR(fb.MoveQueue[selected1[2].index].Commands), sX + sY,  0.020, 0, 0, 0, 0, pathY_X, 0.00, mcACP6D_MOVE_RELATIVE);
					END_IF;

					shuttles[selected1[0].index].command.moveQueue := TRUE;
					shuttles[selected1[1].index].command.moveQueue := TRUE;
					shuttles[selected1[2].index].command.moveQueue := TRUE;
					shuttles[selected1[3].index].command.moveQueue := TRUE;

					IF queueStatus.allDone THEN
						task.SubState := 201;
					ELSIF queueStatus.error THEN
						task.Error.Code := queueStatus.errorID;
						task.State := ACP6D_COMMAND_ERROR;
					END_IF;

				201:
					task.StateInfo := 'Star shift 2';
					// ---------------------------------------------------------------------------------
					IF task.OnStateEntry THEN
						shuttle ACCESS ADR(shuttles[selected1[0].index]);

						shuffle.angle := brmPI_2 * RandValueDINT(3 * 4, 5 * 4);

						brsmemset(ADR(commandQueue), 0, SIZEOF(commandQueue));

						AddCommand6D_waitCmdLb(ADR(commandQueue), shuttle.ID, mcACP6D_SH_WAIT_CMDLB_START, 0, mcACP6D_SH_WAIT_CMDLB_REGULAR);
						AddCommand6D_arcAngularCW(ADR(commandQueue), 2 * 0.24, 3 * 0.24, shuffle.angle, 1.0, 15.0, 0, mcACP6D_MOVE_ABSOLUTE);

						fb.MoveQueue[selected1[1].index].Commands := commandQueue;
						fb.MoveQueue[selected1[2].index].Commands := commandQueue;
						fb.MoveQueue[selected1[3].index].Commands := commandQueue;
					END_IF;

					shuttles[selected1[1].index].command.moveQueue := TRUE;
					shuttles[selected1[2].index].command.moveQueue := TRUE;
					shuttles[selected1[3].index].command.moveQueue := TRUE;

					IF fb.MoveQueue[selected1[1].index].Acknowledge AND fb.MoveQueue[selected1[2].index].Acknowledge AND fb.MoveQueue[selected1[3].index].Acknowledge THEN
						task.SubState := 202;
					ELSIF queueStatus.error THEN
						task.Error.Code := queueStatus.errorID;
						task.State := ACP6D_COMMAND_ERROR;
					END_IF;

				202:
					task.StateInfo := 'Star shift 3';
					// ---------------------------------------------------------------------------------
					IF task.OnStateEntry THEN
						shuttle ACCESS ADR(shuttles[selected1[0].index]);

						AddCommand6D_arcAngularCW(ADR(commandQueue), 2 * 0.24, 3 * 0.24, shuffle.angle, 1.0, 15.0, 0, mcACP6D_MOVE_ABSOLUTE);

						fb.MoveQueue[selected1[0].index].Commands := commandQueue;
					END_IF;

					shuttles[selected1[0].index].command.moveQueue := TRUE;

					IF queueStatus.allDone THEN
						task.SubState := 203;
					ELSIF queueStatus.error THEN
						task.Error.Code := queueStatus.errorID;
						task.State := ACP6D_COMMAND_ERROR;
					END_IF;

				203:
					task.StateInfo := 'Star shift end';
					// ---------------------------------------------------------------------------------
					IF task.OnStateEntry THEN
						brfiShuttleSelect(ADR(shuttles), ADR(selected1), 0, 0.480, 1, 1);

						AddCommand6D_xy(ADR(fb.MoveQueue[selected1[0].index].Commands), sX + sY, positions.shuffle_simple[0].X, positions.shuffle_simple[0].Y, 0, 0, 0, pathDIRECT, 0.00, mcACP6D_MOVE_ABSOLUTE);
						AddCommand6D_xy(ADR(fb.MoveQueue[selected1[1].index].Commands), sX + sY, positions.shuffle_simple[1].X, positions.shuffle_simple[1].Y, 0, 0, 0, pathDIRECT, 0.00, mcACP6D_MOVE_ABSOLUTE);
						AddCommand6D_xy(ADR(fb.MoveQueue[selected1[2].index].Commands), sX + sY, positions.shuffle_simple[2].X, positions.shuffle_simple[2].Y, 0, 0, 0, pathDIRECT, 0.00, mcACP6D_MOVE_ABSOLUTE);
						AddCommand6D_xy(ADR(fb.MoveQueue[selected1[3].index].Commands), sX + sY, positions.shuffle_simple[3].X, positions.shuffle_simple[3].Y, 0, 0, 0, pathDIRECT, 0.00, mcACP6D_MOVE_ABSOLUTE);
					END_IF;

					shuttles[selected1[0].index].command.moveQueue := TRUE;
					shuttles[selected1[1].index].command.moveQueue := TRUE;
					shuttles[selected1[2].index].command.moveQueue := TRUE;
					shuttles[selected1[3].index].command.moveQueue := TRUE;

					IF queueStatus.allDone THEN
						task.SubState := 204;
					ELSIF queueStatus.error THEN
						task.Error.Code := queueStatus.errorID;
						task.State := ACP6D_COMMAND_ERROR;
					END_IF;

				204:
					task.StateInfo := 'End of simple shuffle - move to select';
					// ---------------------------------------------------------------------------------
					IF task.OnStateEntry THEN
						brfiShuttleSelect(ADR(shuttles), ADR(selected1), 0, 0.480, 1, 1);

						AddCommand6D_xy(ADR(fb.MoveQueue[selected1[0].index].Commands), sX + sY, positions.user[2].X, positions.user[2].Y, 1.5, 0, 0, pathDIRECT, 0.00, mcACP6D_MOVE_ABSOLUTE);
						AddCommand6D_xy(ADR(fb.MoveQueue[selected1[1].index].Commands), sX + sY, positions.user[3].X, positions.user[3].Y, 1.5, 0, 0, pathDIRECT, 0.00, mcACP6D_MOVE_ABSOLUTE);
						AddCommand6D_xy(ADR(fb.MoveQueue[selected1[2].index].Commands), sX + sY, positions.user[4].X, positions.user[4].Y, 1.5, 0, 0, pathDIRECT, 0.00, mcACP6D_MOVE_ABSOLUTE);
						AddCommand6D_xy(ADR(fb.MoveQueue[selected1[3].index].Commands), sX + sY, positions.user[5].X, positions.user[5].Y, 1.5, 0, 0, pathDIRECT, 0.00, mcACP6D_MOVE_ABSOLUTE);
					END_IF;

					shuttles[selected1[0].index].command.moveQueue := TRUE;
					shuttles[selected1[1].index].command.moveQueue := TRUE;
					shuttles[selected1[2].index].command.moveQueue := TRUE;
					shuttles[selected1[3].index].command.moveQueue := TRUE;

					IF queueStatus.allDone THEN
						task.State := ACP6D_COMMAND_DONE;
					ELSIF queueStatus.error THEN
						task.Error.Code := queueStatus.errorID;
						task.State := ACP6D_COMMAND_ERROR;
					END_IF;

			END_CASE;

		ACP6D_SHUFFLE_CIRCULAR:
			CASE task.SubState OF
				0:
					task.StateInfo := 'Move shuttles to start position';
					// ---------------------------------------------------------------------------------
					IF task.OnStateEntry THEN
						brfiShuffle(ADR(local.shuttleOrder));

						// Configure shuttle targets
						fb.MoveInPlaneAsync.Parameters.Velocity := 2;
						fb.MoveInPlaneAsync.Parameters.Acceleration := 15;

						fb.MoveInPlaneAsync.Parameters.Mode := mcACP6D_SHUTTLE_SORTED;

						FOR i := 0 TO gMAX_INDEX_SHUTTLE DO
							x := local.shuttleOrder[i];
							fb.MoveInPlaneAsync.Parameters.AsyncPar[i].Shuttle := ADR(shuttles[x].Ref);
							fb.MoveInPlaneAsync.Parameters.AsyncPar[i].X := positions.clockface[i].X;
							fb.MoveInPlaneAsync.Parameters.AsyncPar[i].Y := positions.clockface[i].Y;
						END_FOR;
					END_IF;

					local.actions.substate.moveInPlaneAsync := TRUE;

					IF fb.MoveInPlaneAsync.Done THEN
						task.SubState := 100;
					ELSIF fb.MoveInPlaneAsync.Error THEN
						task.Error.Code := fb.MoveInPlaneAsync.ErrorID;
						task.State := ACP6D_COMMAND_ERROR;
					END_IF;

				100:
					task.StateInfo := 'Add commands to queue';
					// ---------------------------------------------------------------------------------
					IF task.OnStateEntry THEN
						shuttle ACCESS ADR(shuttles[0]);

						shuffle.angle := (brmPI/8) * RandValueDINT(6 * 8, 9 * 8);

						brsmemset(ADR(commandQueue), 0, SIZEOF(commandQueue));

						AddCommand6D_waitCmdLb(ADR(commandQueue), shuttle.ID, mcACP6D_SH_WAIT_CMDLB_START, 0, mcACP6D_SH_WAIT_CMDLB_REGULAR);
						AddCommand6D_arcAngularCW(ADR(commandQueue), 0.48, 0.48, shuffle.angle, 0, 0, 0, mcACP6D_MOVE_ABSOLUTE);

						FOR i := 0 TO gMAX_INDEX_SHUTTLE DO
							fb.MoveQueue[i].Parameters := moveQueueParamDefault;
							fb.MoveQueue[i].Parameters.acceleration := 14.0;
						END_FOR;

						FOR i := 1 TO gMAX_INDEX_SHUTTLE DO
							fb.MoveQueue[i].Commands := commandQueue;
							shuttles[i].command.moveQueue := TRUE;
						END_FOR;
					END_IF

					IF queueStatus.allAcknowledge THEN
						task.SubState := 110;
					ELSIF queueStatus.error THEN
						task.Error.Code := queueStatus.errorID;
						task.State := ACP6D_COMMAND_ERROR;
					END_IF;

				110:
					task.StateInfo := 'Wait to finish circular CW';
					// ---------------------------------------------------------------------------------
					IF task.OnStateEntry THEN
						brsmemset(ADR(commandQueue), 0, SIZEOF(commandQueue));

						AddCommand6D_arcAngularCW(ADR(commandQueue), 0.48, 0.48, shuffle.angle, 0, 0, 0, mcACP6D_MOVE_ABSOLUTE);

						fb.MoveQueue[0].Commands := commandQueue;
						shuttles[0].command.moveQueue := TRUE;
					END_IF

					IF queueStatus.allDone THEN
						task.SubState := 120;
					ELSIF queueStatus.error THEN
						task.Error.Code := queueStatus.errorID;
						task.State := ACP6D_COMMAND_ERROR;
					END_IF;

				120:
					task.StateInfo := 'Add commands to queue';
					// ---------------------------------------------------------------------------------
					IF task.OnStateEntry THEN
						shuttle ACCESS ADR(shuttles[0]);

						shuffle.angle := (brmPI/8) * RandValueDINT(6 * 8, 9 * 8);

						brsmemset(ADR(commandQueue), 0, SIZEOF(commandQueue));

						AddCommand6D_waitCmdLb(ADR(commandQueue), shuttle.ID, mcACP6D_SH_WAIT_CMDLB_START, 0, mcACP6D_SH_WAIT_CMDLB_REGULAR);
						AddCommand6D_arcAngularCCW(ADR(commandQueue), 0.48, 0.48, shuffle.angle, 0, 0, 0, mcACP6D_MOVE_ABSOLUTE);

						FOR i := 1 TO gMAX_INDEX_SHUTTLE DO
							fb.MoveQueue[i].Commands := commandQueue;
							shuttles[i].command.moveQueue := TRUE;
						END_FOR;
					END_IF

					IF queueStatus.allAcknowledge THEN
						task.SubState := 130;
					ELSIF queueStatus.error THEN
						task.Error.Code := queueStatus.errorID;
						task.State := ACP6D_COMMAND_ERROR;
					END_IF;

				130:
					task.StateInfo := 'wait to finish circular CCW';
					// ---------------------------------------------------------------------------------
					IF task.OnStateEntry THEN
						brsmemset(ADR(commandQueue), 0, SIZEOF(commandQueue));

						AddCommand6D_arcAngularCCW(ADR(commandQueue), 0.48, 0.48, shuffle.angle, 0, 0, 0, mcACP6D_MOVE_ABSOLUTE);

						fb.MoveQueue[0].Commands := commandQueue;
						shuttles[0].command.moveQueue := TRUE;
					END_IF

					IF queueStatus.allDone THEN
						task.SubState := 200;
					ELSIF queueStatus.error THEN
						task.Error.Code := queueStatus.errorID;
						task.State := ACP6D_COMMAND_ERROR;
					END_IF;

				200:
					task.StateInfo := 'Move shuttles to kongo line';
					// ---------------------------------------------------------------------------------
					IF task.OnStateEntry THEN
						brfiShuffle(ADR(local.shuttleOrder));

						// Configure shuttle targets
						fb.MoveInPlaneAsync.Parameters.Velocity := 2;
						fb.MoveInPlaneAsync.Parameters.Acceleration := 15;

						fb.MoveInPlaneAsync.Parameters.Mode := mcACP6D_SHUTTLE_SORTED;

						FOR i := 0 TO gMAX_INDEX_SHUTTLE DO
							x := local.shuttleOrder[i];
							fb.MoveInPlaneAsync.Parameters.AsyncPar[i].Shuttle := ADR(shuttles[x].Ref);
							fb.MoveInPlaneAsync.Parameters.AsyncPar[i].X := positions.kongo_lines[i].X;
							fb.MoveInPlaneAsync.Parameters.AsyncPar[i].Y := positions.kongo_lines[i].Y;
						END_FOR;
					END_IF;

					local.actions.substate.moveInPlaneAsync := TRUE;

					IF fb.MoveInPlaneAsync.Done THEN
						task.SubState := 210;
					ELSIF fb.MoveInPlaneAsync.Error THEN
						task.Error.Code := fb.MoveInPlaneAsync.ErrorID;
						task.State := ACP6D_COMMAND_ERROR;
					END_IF;

				210:
					task.StateInfo := 'Move shuttles to start position';
					// ---------------------------------------------------------------------------------
					IF task.OnStateEntry THEN
						brfiShuttleSelect(ADR(shuttles), ADR(selected1), 0, 0, 2 * 0.240, 1);
						brfiShuttleSelect(ADR(shuttles), ADR(selected2), 2 * 0.240, 0, 1, 1);

						AddCommand6D_xy(ADR(commandQueue), sX, 0.240 + 0.120, 0, 0, 0, 1, pathDIRECT, 0, mcACP6D_MOVE_RELATIVE);
						AddCommand6D_arcAngularCCW(ADR(commandQueue), 0, 0.060, brmPI, 0, 0, 1, mcACP6D_MOVE_RELATIVE);
						AddCommand6D_xy(ADR(commandQueue), sX, -0.480, 0, 0, 0, 1, pathDIRECT, 0, mcACP6D_MOVE_RELATIVE);

						AddCommand6D_arcAngularCCW(ADR(commandQueue), 0, -0.060, brmPI, 0, 0, 1, mcACP6D_MOVE_RELATIVE);
						AddCommand6D_xy(ADR(commandQueue), sX, 0.120, 0, 0, 0, 1, pathDIRECT, 0, mcACP6D_MOVE_RELATIVE);
						AddCommand6D_xy(ADR(commandQueue), sX, 0.240 + 0.120, 0, 0, 0, 1, pathDIRECT, 0, mcACP6D_MOVE_RELATIVE);
						AddCommand6D_arcAngularCCW(ADR(commandQueue), 0, 0.060, brmPI, 0, 0, 1, mcACP6D_MOVE_RELATIVE);

						AddCommand6D_xy(ADR(commandQueue), sX, -0.480, 0, 0, 0, 1, pathDIRECT, 0, mcACP6D_MOVE_RELATIVE);
						AddCommand6D_arcAngularCCW(ADR(commandQueue), 0, -0.060, brmPI, 0, 0, 1, mcACP6D_MOVE_RELATIVE);
						AddCommand6D_xy(ADR(commandQueue), sX, 0.240 + 0.120, 0, 0, 0, 1, pathDIRECT, 0, mcACP6D_MOVE_RELATIVE);
						AddCommand6D_arcAngularCCW(ADR(commandQueue), 0, 0.060, brmPI, 0, 0, 1, mcACP6D_MOVE_RELATIVE);

						AddCommand6D_xy(ADR(commandQueue), sX, 2 * 0.240, 0, 0, 0, 0, pathDIRECT, 0, mcACP6D_MOVE_ABSOLUTE);

						FOR i := 0 TO 3 DO
							fb.MoveQueue[selected1[i].index].Commands := commandQueue;
							shuttles[selected1[i].index].command.moveQueue := TRUE;;
						END_FOR;

						brsmemset(ADR(commandQueue), 0, SIZEOF(commandQueue));
						AddCommand6D_xy(ADR(commandQueue), sX, -(0.240 + 0.120), 0, 0, 0, 1, pathDIRECT, 0, mcACP6D_MOVE_RELATIVE);
						AddCommand6D_arcAngularCCW(ADR(commandQueue), 0, -0.060, brmPI, 0, 0, 1, mcACP6D_MOVE_RELATIVE);
						AddCommand6D_xy(ADR(commandQueue), sX, 0.4800, 0, 0, 0, 1, pathDIRECT, 0, mcACP6D_MOVE_RELATIVE);

						AddCommand6D_arcAngularCCW(ADR(commandQueue), 0, 0.060, brmPI, 0, 0, 1, mcACP6D_MOVE_RELATIVE);
						AddCommand6D_xy(ADR(commandQueue), sX, -0.120, 0, 0, 0, 1, pathDIRECT, 0, mcACP6D_MOVE_RELATIVE);
						AddCommand6D_xy(ADR(commandQueue), sX, -(0.240 + 0.120), 0, 0, 0, 1, pathDIRECT, 0, mcACP6D_MOVE_RELATIVE);
						AddCommand6D_arcAngularCCW(ADR(commandQueue), 0, -0.060, brmPI, 0, 0, 1, mcACP6D_MOVE_RELATIVE);

						AddCommand6D_xy(ADR(commandQueue), sX, 0.480, 0, 0, 0, 1, pathDIRECT, 0, mcACP6D_MOVE_RELATIVE);
						AddCommand6D_arcAngularCCW(ADR(commandQueue), 0, 0.060, brmPI, 0, 0, 1, mcACP6D_MOVE_RELATIVE);
						AddCommand6D_xy(ADR(commandQueue), sX, -(0.240 + 0.120), 0, 0, 0, 1, pathDIRECT, 0, mcACP6D_MOVE_RELATIVE);
						AddCommand6D_arcAngularCCW(ADR(commandQueue), 0, -0.060, brmPI, 0, 0, 1, mcACP6D_MOVE_RELATIVE);

						AddCommand6D_xy(ADR(commandQueue), sX, 2 * 0.240, 0, 0, 0, 0, pathDIRECT, 0, mcACP6D_MOVE_ABSOLUTE);

						FOR i := 0 TO 3 DO
							fb.MoveQueue[selected2[i].index].Commands := commandQueue;
							shuttles[selected2[i].index].command.moveQueue := TRUE;;
						END_FOR;

					END_IF

					IF queueStatus.allAcknowledge THEN
						task.SubState := 220;
					ELSIF queueStatus.error THEN
						task.Error.Code := queueStatus.errorID;
						task.State := ACP6D_COMMAND_ERROR;
					END_IF;

				220:
					task.StateInfo := 'Move shuttles';
					// ---------------------------------------------------------------------------------
					IF task.OnStateEntry THEN
						brfiShuttleSelect(ADR(shuttles), ADR(selected1), 0, 0, 4 * 0.240, 2 * 0.240);

						brfiShuttleSelect(ADR(shuttles), ADR(selected2), 2 * 0.240, 0, 1, 1);

						AddCommand6D_xy(ADR(fb.MoveQueue[selected1[0].index].Commands), sX + sY, 0.240, 0.180, 0, 0, 0, pathX_Y, 0, mcACP6D_MOVE_ABSOLUTE);
						AddCommand6D_xy(ADR(fb.MoveQueue[selected1[3].index].Commands), sX + sY, 0.240, 0.300, 0, 0, 0, pathX_Y, 0, mcACP6D_MOVE_ABSOLUTE);

						AddCommand6D_xy(ADR(fb.MoveQueue[selected1[1].index].Commands), sX + sY, 3 * 0.240, 0.180, 0, 0, 0, pathX_Y, 0, mcACP6D_MOVE_ABSOLUTE);
						AddCommand6D_xy(ADR(fb.MoveQueue[selected1[2].index].Commands), sX + sY, 3 * 0.240, 0.300, 0, 0, 0, pathX_Y, 0, mcACP6D_MOVE_ABSOLUTE);

						//
//						brsmemset(ADR(commandQueue), 0, SIZEOF(commandQueue));
//						AddCommand6D_xy(ADR(commandQueue), sX, -(0.240 + 0.120), 0, 0, 0, 1, pathDIRECT, 0, mcACP6D_MOVE_RELATIVE);
//						AddCommand6D_arcAngularCCW(ADR(commandQueue), 0, -0.060, brmPI, 0, 0, 1, mcACP6D_MOVE_RELATIVE);
//						AddCommand6D_xy(ADR(commandQueue), sX, 0.4800, 0, 0, 0, 1, pathDIRECT, 0, mcACP6D_MOVE_RELATIVE);
//
//						AddCommand6D_arcAngularCCW(ADR(commandQueue), 0, 0.060, brmPI, 0, 0, 1, mcACP6D_MOVE_RELATIVE);
//						AddCommand6D_xy(ADR(commandQueue), sX, -0.120, 0, 0, 0, 1, pathDIRECT, 0, mcACP6D_MOVE_RELATIVE);
//						AddCommand6D_xy(ADR(commandQueue), sX, -(0.240 + 0.120), 0, 0, 0, 1, pathDIRECT, 0, mcACP6D_MOVE_RELATIVE);
//						AddCommand6D_arcAngularCCW(ADR(commandQueue), 0, -0.060, brmPI, 0, 0, 1, mcACP6D_MOVE_RELATIVE);
//
//						AddCommand6D_xy(ADR(commandQueue), sX, 0.480, 0, 0, 0, 1, pathDIRECT, 0, mcACP6D_MOVE_RELATIVE);
//						AddCommand6D_arcAngularCCW(ADR(commandQueue), 0, 0.060, brmPI, 0, 0, 1, mcACP6D_MOVE_RELATIVE);
//						AddCommand6D_xy(ADR(commandQueue), sX, -(0.240 + 0.120), 0, 0, 0, 1, pathDIRECT, 0, mcACP6D_MOVE_RELATIVE);
//						AddCommand6D_arcAngularCCW(ADR(commandQueue), 0, -0.060, brmPI, 0, 0, 1, mcACP6D_MOVE_RELATIVE);
//
//						AddCommand6D_xy(ADR(commandQueue), sX, 0.240, 0, 0, 0, 0, pathDIRECT, 0, mcACP6D_MOVE_RELATIVE);

						FOR i := 0 TO gMAX_INDEX_SHUTTLE DO
							shuttles[i].command.moveQueue := TRUE;
						END_FOR;

					END_IF

					IF queueStatus.allAcknowledge THEN
						task.SubState := 240;
					ELSIF queueStatus.error THEN
						task.Error.Code := queueStatus.errorID;
						task.State := ACP6D_COMMAND_ERROR;
					END_IF;

			END_CASE;

		ACP6D_VICTORY:
			CASE task.SubState OF
				0:
					task.StateInfo := 'Move shuttles to start position';
					// ---------------------------------------------------------------------------------
					IF task.OnStateEntry THEN
						// Configure shuttle targets
						fb.MoveInPlaneAsync.Parameters.Velocity := 2;
						fb.MoveInPlaneAsync.Parameters.Acceleration := 15;

						fb.MoveInPlaneAsync.Parameters.Mode := mcACP6D_SHUTTLE_UNSORTED;

						FOR i := 0 TO gMAX_INDEX_SHUTTLE DO
							fb.MoveInPlaneAsync.Parameters.AsyncPar[i].Shuttle := ADR(shuttles[i].Ref);
							fb.MoveInPlaneAsync.Parameters.AsyncPar[i].X := positions.dance[i].X;
							fb.MoveInPlaneAsync.Parameters.AsyncPar[i].Y := positions.dance[i].Y;
						END_FOR;
					END_IF;

					local.actions.substate.moveInPlaneAsync := TRUE;

					IF fb.MoveInPlaneAsync.Done THEN
						task.State := ACP6D_COMMAND_DONE;
					ELSIF fb.MoveInPlaneAsync.Error THEN
						task.Error.Code := fb.MoveInPlaneAsync.ErrorID;
						task.State := ACP6D_COMMAND_ERROR;
					END_IF;
			END_CASE

		ACP6D_COMMAND_DONE:
			task.StateInfo := 'Command done';
			// ---------------------------------------------------------------------------------
			// Check that all commands are reset
			IF brsmemcmp(ADR(no_command), ADR(task.Input.Command), SIZEOF(no_command)) = 0 THEN
				task.State := ACP6D_IDLE;
			END_IF;

		ACP6D_COMMAND_ERROR:
			task.StateInfo := 'Command failed';
			// ---------------------------------------------------------------------------------
			// Check that all commands are reset
			IF brsmemcmp(ADR(no_command), ADR(task.Input.Command), SIZEOF(no_command)) = 0 THEN
				brsmemset(ADR(task.Error), 0, SIZEOF(task.Error));
				task.State := ACP6D_IDLE;
			END_IF;

		ACP6D_ERROR:
			CASE task.SubState OF
				0:
					task.StateInfo := 'Wait for error acknowledge command';
					// ---------------------------------------------------------------------------------
					local.actions.state.cyclicModeRequest := a6dCYCLIC_DISABLED;

					IF task.Error.Acknowledge THEN
						task.SubState := 10;
					END_IF;

				10:
					task.StateInfo := 'Resetting assembly errors';
					// ---------------------------------------------------------------------------------
					local.actions.substate.assemblyReset := TRUE;
					IF task.Output.AssemblyInfo.AssemblyState <> mcACP6D_ERRORSTOP THEN
						brsmemset(ADR(task.Error), 0, SIZEOF(task.Error));
						task.State := ACP6D_INITIALIZE;
					END_IF;
			END_CASE;
	END_CASE // End of main task logic

	task.Error.Acknowledge := FALSE;

	// Detect state change events
	// =================================================================================================================
	task.OnStateEntry := (task.State <> local.lastState) OR (task.SubState <> local.lastSubState);

	IF task.State <> local.lastState THEN
		IF (task.State = ACP6D_ERROR) OR (task.State = ACP6D_COMMAND_ERROR) THEN
	  		task.Error.State := task.State;
			task.Error.SubState := task.SubState;
		END_IF;

		task.SubState := 0;
		local.lastState := task.State;
		brsmemset(ADR(local.actions.state), 0, SIZEOF(local.actions.state));
		brsmemset(ADR(local.actions.substate), 0, SIZEOF(local.actions.substate));
		task.StateInfo := '';

		// Reset to default on every major task change
		moveQueueParamTask := moveQueueParamDefault;
	END_IF

	// Reset current state actions also when substate changes
	IF task.SubState <> local.lastSubState THEN
		local.lastSubState := task.SubState;
		brsmemset(ADR(local.actions.substate), 0, SIZEOF(local.actions.substate));
		task.StateInfo := '';
	END_IF

	IF task.OnStateEntry THEN
		brsmemset(ADR(commandQueue), 0, SIZEOF(commandQueue));

		IF task.State <> ACP6D_COMMAND_ERROR THEN
			FOR i := 0 TO gMAX_INDEX_SHUTTLE DO
				brsmemset(ADR(shuttles[i].command), 0, SIZEOF(shuttles[i].command));
				brsmemset(ADR(fb.MoveInPlaneAsync.Parameters.AsyncPar), 0, SIZEOF(fb.MoveInPlaneAsync.Parameters.AsyncPar));
				brsmemset(ADR(fb.MoveQueue[i].Commands), 0, SIZEOF(fb.MoveQueue[i].Commands));
			END_FOR;
		END_IF;
	END_IF;

	// Function calls
	// =================================================================================================================
	fb.AssemblyReadInfo.Assembly := ADR(gAssembly6D_1);
	fb.AssemblyReadInfo();

	fb.AssemblyPowerOn.Assembly := ADR(gAssembly6D_1);
	fb.AssemblyPowerOn.Execute := local.actions.substate.assemblyPowerOn;
	fb.AssemblyPowerOn();

	fb.AssemblyPowerOff.Assembly := ADR(gAssembly6D_1);
	fb.AssemblyPowerOff.Execute := local.actions.substate.assemblyPowerOff;
	fb.AssemblyPowerOff();

	fb.AssemblyReset.Assembly := ADR(gAssembly6D_1);
	fb.AssemblyReset.Execute := local.actions.substate.assemblyReset;
	fb.AssemblyReset();

	fb.AssemblyGetShuttle.Assembly := ADR(gAssembly6D_1);
	fb.AssemblyGetShuttle.Enable := local.actions.state.assemblyGetShuttles;
	fb.AssemblyGetShuttle.Next := local.actions.state.assemblyGetNextShuttle;
	fb.AssemblyGetShuttle();

	fb.MoveInPlaneAsync.Assembly := ADR(gAssembly6D_1);
	fb.MoveInPlaneAsync.Execute := local.actions.substate.moveInPlaneAsync;
	fb.MoveInPlaneAsync();

	fb.TON_delay.IN := local.actions.substate.delay;
	fb.TON_delay();

	fb.assemblyStop.Assembly := ADR(gAssembly6D_1);
	fb.assemblyStop.Execute := local.actions.substate.assemblyStop;
	fb.assemblyStop();

	fb.assemblyGetVirtualSh.Assembly := ADR(gAssembly6D_1);
	fb.assemblyGetVirtualSh();

	fb.virtualShCreate.Assembly := ADR(gAssembly6D_1);
	fb.virtualShCreate.Execute := local.actions.substate.createShuttleVirtual;
	fb.virtualShCreate();

	// Call shuttle functions
	FOR i := 0 TO gMAX_INDEX_SHUTTLE DO
		fb.Move6D[i].Shuttle := ADR(shuttles[i].Ref);
		fb.Move6D[i].Execute := shuttles[i].command.move6D;
		fb.Move6D[i]();

		fb.MoveQueue[i].Shuttle := ADR(shuttles[i].Ref);
		fb.MoveQueue[i].Execute := shuttles[i].command.moveQueue;
		fb.MoveQueue[i]();
	END_FOR;

	// 6D Cyclic channel handling
	// =================================================================================================================
	acCyclicChannelHandling;

	// Update shuttle statuses by polling them one by one
	// =================================================================================================================
    acShuttleStatusPolling;

	// Move Queue status handling
	// =================================================================================================================
	acMoveQueueStatusHandling;

	// Generate random numbers
	// =================================================================================================================
	random.delays[random.delaysIndex] := RandValueREAL(100, 2000) / 1000;
	random.delaysIndex := random.delaysIndex + 1;
	IF random.delaysIndex > gMAX_INDEX_SHUTTLE THEN
		random.delaysIndex := 0;
	END_IF;

	random.shuffleSequence[random.shuffleSequenceIndex] := RandValueDINT(-1000, 1000) MOD 5;
	random.shuffleSequenceIndex := random.shuffleSequenceIndex + 1;
	IF random.shuffleSequenceIndex > gMAX_INDEX_SHUFFLE THEN
		random.shuffleSequenceIndex := 0;
	END_IF;

	// Task outputs
	// =================================================================================================================
	task.Output.AssemblyInfo := fb.AssemblyReadInfo.AssemblyInfo;
	task.Output.Status.CommandDone := (task.State = ACP6D_COMMAND_DONE);
	task.Error.Active := (task.State = ACP6D_ERROR) OR (task.State = ACP6D_COMMAND_ERROR);

	task.Output.ShuttleUserSelected.X := shuttles[task.Output.ShuttleUserSelected.index].position.value.X;
	task.Output.ShuttleUserSelected.Y := shuttles[task.Output.ShuttleUserSelected.index].position.value.Y;

	task.Output.ShuttleWithPayload.X := shuttles[task.Output.ShuttleWithPayload.index].position.value.X;
	task.Output.ShuttleWithPayload.Y := shuttles[task.Output.ShuttleWithPayload.index].position.value.Y;

END_PROGRAM

PROGRAM _EXIT

END_PROGRAM
```

#### local.typ
```iecst
TYPE
	Acp6DActionsType : 	STRUCT
		task : Acp6DTaskActionsType; (*Task actions are not automatically reset*)
		state : Acp6DStateActionsType; (*State actions are automatically reset whenever major task changes*)
		substate : Acp6DSubstateActionsType; (*Substate actions are automatically reset whenever major or substate changes*)
	END_STRUCT;
	Acp6DFbType : 	STRUCT
		AssemblyReadInfo : MC_BR_AsmReadInfo_Acp6D;
		AssemblyPowerOn : MC_BR_AsmPowerOn_Acp6D;
		AssemblyPowerOff : MC_BR_AsmPowerOff_Acp6D;
		AssemblyReset : MC_BR_AsmReset_Acp6D;
		AssemblyGetShuttle : MC_BR_AsmGetShuttle_Acp6D;
		assemblyStop : MC_BR_AsmStop_Acp6D;
		MoveInPlaneAsync : MC_BR_MoveInPlaneAsync_Acp6D;
		TON_delay : TON;
		Move6D : ARRAY[0..gMAX_INDEX_SHUTTLE]OF MC_BR_Move6D_Acp6D;
		ReadCyclicForce : ARRAY[0..gMAX_INDEX_SHUTTLE]OF MC_BR_ReadCyclicForce_Acp6D;
		ReadCyclicPosition : ARRAY[0..gMAX_INDEX_SHUTTLE]OF MC_BR_ReadCyclicPosition_Acp6D;
		MoveCyclicPosition : ARRAY[0..gMAX_INDEX_SHUTTLE]OF MC_BR_MoveCyclicPosition_Acp6D;
		MoveQueue : ARRAY[0..gMAX_INDEX_SHUTTLE]OF brfi6DMoveQueue;
		ShGetInfo : MC_BR_ShGetInfo_Acp6D;
		virtualShCreate : MC_BR_VirtualShCreate_Acp6D;
		assemblyGetVirtualSh : MC_BR_AsmGetVirtualSh_Acp6D;
	END_STRUCT;
	Acp6DHmiType : 	STRUCT
		isRunning : BOOL;
	END_STRUCT;
	Acp6DLocalType : 	STRUCT
		lastState : DINT;
		lastSubState : DINT;
		actions : Acp6DActionsType;
		allValid : BOOL;
		measurement_index : DINT;
		targetPos : ARRAY[0..gMAX_INDEX_SHUTTLE]OF McAcp6DShPositionType;
		shuttleOrder : ARRAY[0..gMAX_INDEX_SHUTTLE]OF DINT;
		Fz_highest : REAL;
		executing : BOOL;
		selectedCount : DINT;
		virtualShuttleCount : DINT;
	END_STRUCT;
	Acp6DTaskActionsType : 	STRUCT
		dummy : BOOL;
	END_STRUCT;
	Acp6DStateActionsType : 	STRUCT
		assemblyGetShuttles : BOOL;
		assemblyGetNextShuttle : BOOL;
		cyclicModeRequest : Acp6DCyclicModeEnum;
	END_STRUCT;
	Acp6DSubstateActionsType : 	STRUCT
		assemblyPowerOff : BOOL;
		assemblyPowerOn : BOOL;
		assemblyReset : BOOL;
		assemblyStop : BOOL;
		createShuttleVirtual : BOOL;
		moveInPlaneAsync : BOOL;
		delay : BOOL;
	END_STRUCT;
	Acp6DTablePositionType : 	STRUCT
		home : ARRAY[0..gMAX_INDEX_SHUTTLE]OF McAcp6DShPositionType;
		user : ARRAY[0..gMAX_INDEX_SHUTTLE]OF McAcp6DShPositionType;
		side : ARRAY[0..gMAX_INDEX_SHUTTLE]OF McAcp6DShPositionType;
		pickup : ARRAY[0..gMAX_INDEX_SHUTTLE]OF McAcp6DShPositionType;
		shuffle : ARRAY[0..gMAX_INDEX_SHUTTLE]OF McAcp6DShPositionType;
		clockface : ARRAY[0..gMAX_INDEX_SHUTTLE]OF McAcp6DShPositionType;
		dance : ARRAY[0..gMAX_INDEX_SHUTTLE]OF McAcp6DShPositionType;
		shuffle_simple : ARRAY[0..gMAX_INDEX_SHUTTLE]OF McAcp6DShPositionType;
		kongo_lines : ARRAY[0..gMAX_INDEX_SHUTTLE]OF McAcp6DShPositionType;
	END_STRUCT;
END_TYPE

(**)

TYPE
	Acp6DCyclicChannelsType : 	STRUCT
		mode : Acp6DCyclicModeEnum;
		allChannelsReleased : BOOL;
		allPositionsValid : BOOL;
		allForceValuesValid : BOOL;
		allControlReady : BOOL;
	END_STRUCT;
	Acp6DCyclicModeEnum :
		(
		a6dCYCLIC_DISABLED := -1,
		a6dCYCLIC_READ_POSITION,
		a6dCYCLIC_READ_FORCE,
		a6dCYCLIC_MOVE_POSITION,
		a6dCYCLIC_RELEASE_CHANNELS
		);
END_TYPE

(**)

TYPE
	Acp6DMoveQueueStatusType : 	STRUCT
		executing : BOOL;
		allDone : BOOL;
		allAcknowledge : BOOL;
		error : BOOL;
		errorID : DINT;
	END_STRUCT;
END_TYPE

(**)

TYPE
	Acp6DShuttleStatusPollType : 	STRUCT
		state : DINT;
		index : DINT;
		allValid : BOOL;
		allIdle : BOOL;
	END_STRUCT;
	Acp6DShuffleType : 	STRUCT
		invertedMove : BOOL;
		invertedDirection : DINT;
		randNum : DINT;
		payloadPos : DINT;
		angle : REAL;
		step : DINT;
		sequence : ARRAY[0..gMAX_INDEX_SHUFFLE]OF DINT;
	END_STRUCT;
	Acp6DRandomType : 	STRUCT
		delaysIndex : DINT;
		delays : ARRAY[0..gMAX_INDEX_SHUTTLE]OF REAL;
		shuffleSequenceIndex : DINT;
		shuffleSequence : ARRAY[0..gMAX_INDEX_SHUFFLE]OF DINT;
	END_STRUCT;
END_TYPE
```

#### local.var
```iecst
VAR
	refMoveQueue : REFERENCE TO brfi6DMoveQueue;
	task : REFERENCE TO Acp6DType;
	local : Acp6DLocalType;
	fb : Acp6DFbType;
	hmi : Acp6DHmiType;
	i : DINT;
	x : DINT;
	no_command : Acp6DInputCommandType;
	shuttle : REFERENCE TO Acp6dShuttleType;
	commandQueue : ARRAY[0..gMAX_INDEX_TARGETS] OF brfi6DMoveQueueCommandType;
	cyclic : Acp6DCyclicChannelsType;
	queueStatus : Acp6DMoveQueueStatusType;
	shuttleStatus : Acp6DShuttleStatusPollType;
	moveQueueParamDefault : brfi6DMoveQueueParamType;
	moveQueueParamTask : brfi6DMoveQueueParamType;
	shuffle : Acp6DShuffleType;
	selected1 : ARRAY[0..gMAX_INDEX_SHUTTLE] OF brfiShuttleSelectionType;
	selected2 : ARRAY[0..gMAX_INDEX_SHUTTLE] OF brfiShuttleSelectionType;
	random : Acp6DRandomType;
END_VAR
(**)
(*ACOPOS 6D*)
VAR
	shuttles : ARRAY[0..gMAX_INDEX_SHUTTLE] OF Acp6dShuttleType; (*Global shuttle list*)
	shuttlesVirtual : ARRAY[0..gMAX_INDEX_SHUTTLE_VIRTUAL] OF Mc6DShuttleType; (*Global shuttle list*)
	positions : Acp6DTablePositionType;
	test : brfiSunPlanet;
END_VAR
```

#### Action.st
```iecst
ACTION acInitializePositions:

	// ---------------------------------------------------------------------------------------
	FOR i := 0 TO gMAX_INDEX_SHUTTLE DO
		positions.home[i].X := i MOD 4 * 0.120 + 0.240 + 0.060;
		IF i < 4 THEN
			positions.home[i].Y := 0.180 + 0.240;
		ELSE
			positions.home[i].Y := 0.180 + 0.240 + 0.120;
		END_IF;
	END_FOR;

	// ---------------------------------------------------------------------------------------
	FOR i := 0 TO gMAX_INDEX_SHUTTLE DO
		positions.user[i].X := i * 0.120 + 0.060;
		positions.user[i].Y := 1 * 0.240 + 0.120;
	END_FOR;

	// ---------------------------------------------------------------------------------------
	FOR i := 0 TO gMAX_INDEX_SHUTTLE DO
		positions.side[i].X := 4 * 0.240 - 0.060;
		positions.side[i].Y := 0.060 + i * 0.120;
	END_FOR;

	// ---------------------------------------------------------------------------------------
	FOR i := 0 TO gMAX_INDEX_SHUTTLE DO
		IF (i MOD 2) = 0 THEN
			positions.shuffle[i].X := 0.480 + COS(DINT_TO_REAL(i) * 45.0 * brmPI/180.0) * 0.420;
			positions.shuffle[i].Y := 0.480 + SIN(DINT_TO_REAL(i) * 45.0 * brmPI/180.0) * 0.420;
		ELSE
			positions.shuffle[i].X := 0.480 + COS(DINT_TO_REAL(i) * 45.0 * brmPI/180.0) * 0.240;
			positions.shuffle[i].Y := 0.480 + SIN(DINT_TO_REAL(i) * 45.0 * brmPI/180.0) * 0.240;
		END_IF;
	END_FOR;

	// ---------------------------------------------------------------------------------------
	FOR i := 0 TO gMAX_INDEX_SHUTTLE DO
		positions.clockface[i].X := 0.480 + COS(DINT_TO_REAL(i) * 45.0 * brmPI/180.0) * 0.300;
		positions.clockface[i].Y := 0.480 + SIN(DINT_TO_REAL(i) * 45.0 * brmPI/180.0) * 0.300;
	END_FOR;

	// ---------------------------------------------------------------------------------------
	positions.dance[0].X := 0 * 0.24 + 0.12;
	positions.dance[0].Y := 0 * 0.24 + 0.12;
	positions.dance[1].X := 3 * 0.24 + 0.12;
	positions.dance[1].Y := 0 * 0.24 + 0.12;
	positions.dance[2].X := 0 * 0.24 + 0.12;
	positions.dance[2].Y := 3 * 0.24 + 0.12;
	positions.dance[3].X := 3 * 0.24 + 0.12;
	positions.dance[3].Y := 3 * 0.24 + 0.12;

	positions.dance[4].X := 1 * 0.24 + 0.12;
	positions.dance[4].Y := 1 * 0.24 + 0.12;
	positions.dance[5].X := 1 * 0.24 + 0.12;
	positions.dance[5].Y := 2 * 0.24 + 0.12;
	positions.dance[6].X := 2 * 0.24 + 0.12;
	positions.dance[6].Y := 1 * 0.24 + 0.12;
	positions.dance[7].X := 2 * 0.24 + 0.12;
	positions.dance[7].Y := 2 * 0.24 + 0.12;

	// ---------------------------------------------------------------------------------------
	positions.pickup[0].X := 0.480;
	positions.pickup[0].Y := 0.480;

	FOR i := 1 TO gMAX_INDEX_SHUTTLE DO
		positions.pickup[i].X := 0.480 + COS(DINT_TO_REAL(i - 1) * (180/6) * brmPI/180.0) * 0.360;
		positions.pickup[i].Y := 0.310 + SIN(DINT_TO_REAL(i - 1) * (180/6) * brmPI/180.0) * 0.360;
	END_FOR

	// Simple shuffle
	// ---------------------------------------------------------------------------------------
	FOR i := 0 TO gMAX_INDEX_SHUTTLE DO
		IF i < 4 THEN
			positions.shuffle_simple[i].X := 0.120 + i * 0.240;
			positions.shuffle_simple[i].Y := 3 * 0.240;
		ELSE
			positions.shuffle_simple[i].X := 0.300 + (i MOD 4) * 0.120;
			positions.shuffle_simple[i].Y := 0.120;
		END_IF;
	END_FOR;

	// Kongo lines
	// ---------------------------------------------------------------------------------------
	FOR i := 0 TO gMAX_INDEX_SHUTTLE DO
		IF i < 4 THEN
			positions.kongo_lines[i].X := 0.120 + 0.240;
			positions.kongo_lines[i].Y := 0.060 + i * 0.240;
		ELSE
			positions.kongo_lines[i].X := 2 * 0.240 + 0.120;
			positions.kongo_lines[i].Y := 0.180 + (i MOD 4) * 0.240;
		END_IF;
	END_FOR;

END_ACTION

ACTION acClearTargetQueues :

	FOR i := 0 TO gMAX_INDEX_SHUTTLE DO
		brsmemset(ADR(fb.Move6DQueue[i].Targets), 0, SIZEOF(fb.Move6DQueue[i].Targets));
		brsmemset(ADR(fb.MoveXYQueue[i].Targets), 0, SIZEOF(fb.MoveXYQueue[i].Targets));
	END_FOR;

END_ACTION

ACTION acCyclicChannelHandling :

	FOR i := 0 TO gMAX_INDEX_SHUTTLE DO
		fb.ReadCyclicPosition[i].Enable := FALSE;
		shuttles[i].position.isValid := FALSE;

		fb.ReadCyclicForce[i].Enable := FALSE;
		shuttles[i].force.isValid := FALSE;

		fb.MoveCyclicPosition[i].Enable := FALSE;
		shuttles[i].moveCyclicActive := FALSE;
	END_FOR;

	// set global statuses so states can use them if required
	cyclic.allPositionsValid := TRUE;
	cyclic.allForceValuesValid := TRUE;
	cyclic.allControlReady := TRUE;
	cyclic.allChannelsReleased := FALSE;

	FOR i := 0 TO gMAX_INDEX_SHUTTLE DO
		IF NOT fb.ReadCyclicPosition[i].Valid THEN
			cyclic.allPositionsValid := FALSE;
		END_IF;

		IF NOT fb.ReadCyclicForce[i].Valid THEN
			cyclic.allForceValuesValid := FALSE;
		END_IF;

		IF NOT fb.MoveCyclicPosition[i].Valid THEN
			cyclic.allControlReady := FALSE;
		END_IF;
	END_FOR;

	CASE cyclic.mode OF
		a6dCYCLIC_DISABLED:
			// ---------------------------------------------------------------------------------
			CASE local.actions.state.cyclicModeRequest OF
				a6dCYCLIC_READ_POSITION:
					cyclic.mode := a6dCYCLIC_READ_POSITION;
				a6dCYCLIC_READ_FORCE:
					cyclic.mode := a6dCYCLIC_READ_FORCE;
				a6dCYCLIC_MOVE_POSITION:
					cyclic.mode := a6dCYCLIC_MOVE_POSITION;
			END_CASE;

		a6dCYCLIC_RELEASE_CHANNELS:
			// ---------------------------------------------------------------------------------
			cyclic.allChannelsReleased := TRUE;

			FOR i := 0 TO gMAX_INDEX_SHUTTLE DO
				IF fb.ReadCyclicPosition[i].Busy OR fb.ReadCyclicForce[i].Busy OR fb.MoveCyclicPosition[i].Busy THEN
					cyclic.allChannelsReleased := FALSE;
				END_IF;
			END_FOR;

			IF cyclic.allChannelsReleased THEN
				cyclic.mode := a6dCYCLIC_DISABLED;
			END_IF;

		a6dCYCLIC_READ_POSITION:
			// ---------------------------------------------------------------------------------
			IF local.actions.state.cyclicModeRequest <> a6dCYCLIC_READ_POSITION THEN
				cyclic.mode := a6dCYCLIC_RELEASE_CHANNELS;
			ELSE
				FOR i := 0 TO gMAX_INDEX_SHUTTLE DO
					fb.ReadCyclicPosition[i].Enable := TRUE;

					IF fb.ReadCyclicPosition[i].Valid THEN
						shuttles[i].position.value := fb.ReadCyclicPosition[i].CyclicPosition;
						shuttles[i].position.isValid := TRUE;
					END_IF;
				END_FOR;
			END_IF;

		a6dCYCLIC_READ_FORCE:
			// ---------------------------------------------------------------------------------
			IF local.actions.state.cyclicModeRequest <> a6dCYCLIC_READ_FORCE THEN
				cyclic.mode := a6dCYCLIC_RELEASE_CHANNELS;
			ELSE
				FOR i := 0 TO gMAX_INDEX_SHUTTLE DO
					fb.ReadCyclicForce[i].Enable := TRUE;
					fb.ReadCyclicForce[i]();

					IF fb.ReadCyclicForce[i].Valid THEN
						shuttles[i].force.value := fb.ReadCyclicForce[i].CyclicForce;
						shuttles[i].force.isValid := TRUE;
					END_IF;
				END_FOR;
			END_IF;

		a6dCYCLIC_MOVE_POSITION:
			// ---------------------------------------------------------------------------------
			IF local.actions.state.cyclicModeRequest <> a6dCYCLIC_MOVE_POSITION THEN
				cyclic.mode := a6dCYCLIC_RELEASE_CHANNELS;
			ELSE
				FOR i := 0 TO gMAX_INDEX_SHUTTLE DO
					fb.MoveCyclicPosition[i].Enable := TRUE;
					fb.MoveCyclicPosition[i]();

					IF fb.MoveCyclicPosition[i].Valid THEN
						shuttles[i].moveCyclicActive := TRUE;
					END_IF;
				END_FOR;
			END_IF;
	END_CASE;

	FOR i := 0 TO gMAX_INDEX_SHUTTLE DO
		fb.ReadCyclicPosition[i].Shuttle := ADR(shuttles[i].Ref);
		fb.ReadCyclicPosition[i]();

		fb.ReadCyclicForce[i].Shuttle := ADR(shuttles[i].Ref);
		fb.ReadCyclicForce[i]();

		fb.MoveCyclicPosition[i].Shuttle := ADR(shuttles[i].Ref);
		fb.MoveCyclicPosition[i]();
	END_FOR;

END_ACTION

ACTION acShuttleStatusPolling :

	shuttleStatus.allValid := TRUE;

	FOR i := 0 TO gMAX_INDEX_SHUTTLE DO
		IF (shuttles[i].Ref.controlif > 0) AND (NOT shuttles[i].status.isValid) THEN
			shuttleStatus.allValid := FALSE;
		END_IF;
	END_FOR;

	shuttleStatus.allIdle := TRUE;

	IF shuttleStatus.allValid THEN
		FOR i := 0 TO gMAX_INDEX_SHUTTLE DO
			IF shuttles[i].status.state <> mcACP6D_SH_STATE_IDLING THEN
				shuttleStatus.allIdle := FALSE;
			END_IF;
		END_FOR;
	ELSE
		shuttleStatus.allIdle := FALSE;
	END_IF;

	CASE shuttleStatus.state OF
		0:
			// ---------------------------------------------------------------------------------
			CASE task.Output.AssemblyInfo.AssemblyState OF
				mcACP6D_INVALID_CONFIGURATION,
				mcACP6D_STARTUP:
					// Wait
				ELSE
					shuttleStatus.state := 10;
					shuttleStatus.index := 0;
			END_CASE;

			FOR i := 0 TO gMAX_INDEX_SHUTTLE DO
				brsmemset(ADR(shuttles[i].status), 0, SIZEOF(shuttles[i].status));
			END_FOR;

			fb.ShGetInfo.Execute := FALSE;

		10:
			// ---------------------------------------------------------------------------------
			CASE task.Output.AssemblyInfo.AssemblyState OF
				mcACP6D_INVALID_CONFIGURATION:
				mcACP6D_STARTUP:
					shuttleStatus.state := 0;
			END_CASE;

			fb.ShGetInfo.Execute := TRUE;

			IF fb.ShGetInfo.Done THEN
				shuttles[shuttleStatus.index].status.isValid := TRUE;
				shuttles[shuttleStatus.index].status.state := fb.ShGetInfo.ShuttleInfo.State;
				shuttleStatus.index := shuttleStatus.index + 1;

			ELSIF fb.ShGetInfo.Error THEN
				brsmemset(ADR(shuttles[shuttleStatus.index].status), 0, SIZEOF(shuttles[shuttleStatus.index].status));
				shuttleStatus.index := shuttleStatus.index + 1;
			END_IF;
	END_CASE;

	IF shuttleStatus.index > gMAX_INDEX_SHUTTLE THEN
		shuttleStatus.index := 0;
	END_IF;

	fb.ShGetInfo.Shuttle := ADR(shuttles[shuttleStatus.index].Ref);
	fb.ShGetInfo();

END_ACTION

ACTION acMoveQueueStatusHandling:

	queueStatus.executing := FALSE;

	FOR i := 0 TO gMAX_INDEX_SHUTTLE DO
		IF fb.MoveQueue[i].Execute THEN
			queueStatus.executing := TRUE;
		END_IF;
	END_FOR;

	IF NOT queueStatus.executing THEN
		queueStatus.allDone := FALSE;
		queueStatus.allAcknowledge := FALSE;
		queueStatus.error := FALSE;
	ELSE
		queueStatus.allDone := TRUE;
		queueStatus.allAcknowledge := TRUE;
		queueStatus.error := FALSE;

		FOR i := 0 TO gMAX_INDEX_SHUTTLE DO
			IF fb.MoveQueue[i].Execute AND (NOT fb.MoveQueue[i].Done) THEN
				queueStatus.allDone := FALSE;
			END_IF;

			IF fb.MoveQueue[i].Execute AND (NOT fb.MoveQueue[i].Acknowledge) THEN
				queueStatus.allAcknowledge := FALSE;
			END_IF;

			IF fb.MoveQueue[i].Execute AND fb.MoveQueue[i].Error THEN
				queueStatus.error := TRUE;
				queueStatus.errorID := fb.MoveQueue[i].ErrorID;
			END_IF;
		END_FOR;
	END_IF;

END_ACTION
```

### Program Logical/Conf6D (ANSIC)
